	UF : 7, UT : 3,	CONFIG : 'F U T, 0, 0, 0',
	X =   -14.765  mm,	Y =   389.269  mm,	Z =     0.000  mm,
	W =  -167.358 deg,	P =     0.000 deg,	R =  -162.799 deg
};
P[92]{
   GP1:
	UF : 7, UT : 3,	CONFIG : 'F U T, 0, 0, 0',
	X =   -39.441  mm,	Y =   387.542  mm,	Z =     0.000  mm,
	W =  -167.357 deg,	P =     0.000 deg,	R =  -159.120 deg
};
P[93]{
   GP1:
	UF : 7, UT : 3,	CONFIG : 'F U T, 0, 0, 0',
	X =   -63.911  mm,	Y =   384.264  mm,	Z =     0.000  mm,
	W =  -167.357 deg,	P =     0.000 deg,	R =  -155.406 deg
};
P[94]{
   GP1:
	UF : 7, UT : 3,	CONFIG : 'F U T, 0, 0, 0',
	X =   -88.261  mm,	Y =   379.415  mm,	Z =     0.000  mm,
	W =  -167.357 deg,	P =    -0.001 deg,	R =  -151.728 deg
};
P[95]{
   GP1:
	UF : 7, UT : 3,	CONFIG : 'F U T, 0, 0, 0',
	X =  -112.432  mm,	Y =   372.971  mm,	Z =     0.000  mm,
	W =  -167.357 deg,	P =    -0.001 deg,	R =  -148.074 deg
};
P[96]{
   GP1:
	UF : 7, UT : 3,	CONFIG : 'F U T, 0, 0, 0',
	X =  -136.150  mm,	Y =   364.985  mm,	Z =     0.000  mm,
	W =  -167.357 deg,	P =    -0.002 deg,	R =  -144.425 deg
};
P[97]{
   GP1:
	UF : 7, UT : 3,	CONFIG : 'F U T, 0, 0, 0',
	X =  -159.308  mm,	Y =   355.490  mm,	Z =     0.000  mm,
	W =  -167.357 deg,	P =    -0.002 deg,	R =  -140.788 deg
};
P[98]{
   GP1:
	UF : 7, UT : 3,	CONFIG : 'F U T, 0, 0, 0',
	X =  -181.924  mm,	Y =   344.465  mm,	Z =     0.001  mm,
	W =  -167.357 deg,	P =    -0.003 deg,	R =  -137.121 deg
};
P[99]{
   GP1:
	UF : 7, UT : 3,	CONFIG : 'F U T, 0, 0, 0',
	X =  -201.161  mm,	Y =   333.583  mm,	Z =     0.001  mm,
	W =  -167.339 deg,	P =    -0.003 deg,	R =  -133.813 deg
};
P[100]{
   GP1:
	UF : 7, UT : 3,	CONFIG : 'F U T, 0, 0, 0',
	X =  -219.916  mm,	Y =   321.550  mm,	Z =     0.002  mm,
	W =  -167.321 deg,	P =    -0.006 deg,	R =  -130.535 deg
};
P[101]{
   GP1:
	UF : 7, UT : 3,	CONFIG : 'F U T, 0, 0, 0',
	X =  -238.197  mm,	Y =   308.239  mm,	Z =     0.003  mm,
	W =  -167.303 deg,	P =    -0.011 deg,	R =  -127.314 deg
};
P[102]{
   GP1:
	UF : 7, UT : 3,	CONFIG : 'F U T, 0, 0, 0',
	X =  -255.186  mm,	Y =   294.327  mm,	Z =     0.005  mm,
	W =  -167.286 deg,	P =    -0.018 deg,	R =  -123.984 deg
};
P[103]{
   GP1:
	UF : 7, UT : 3,	CONFIG : 'F U T, 0, 0, 0',
	X =  -271.779  mm,	Y =   279.082  mm,	Z =     0.007  mm,
	W =  -167.270 deg,	P =    -0.026 deg,	R =  -120.751 deg
};
P[104]{
   GP1:
	UF : 7, UT : 3,	CONFIG : 'F U T, 0, 0, 0',
	X =  -286.942  mm,	Y =   263.454  mm,	Z =     0.009  mm,
	W =  -167.255 deg,	P =    -0.037 deg,	R =  -117.421 deg
};
P[105]{
   GP1:
	UF : 7, UT : 3,	CONFIG : 'F U T, 0, 0, 0',
	X =  -298.890  mm,	Y =   249.815  mm,	Z =     0.013  mm,
	W =  -167.199 deg,	P =    -0.062 deg,	R =  -114.916 deg
};
P[106]{
   GP1:
	UF : 7, UT : 3,	CONFIG : 'F U T, 0, 0, 0',
	X =  -309.583  mm,	Y =   236.436  mm,	Z =     0.019  mm,
	W =  -167.149 deg,	P =    -0.092 deg,	R =  -112.269 deg
};
P[107]{
   GP1:
	UF : 7, UT : 3,	CONFIG : 'F U T, 0, 0, 0',
	X =  -320.386  mm,	Y =   221.580  mm,	Z =     0.036  mm,
	W =  -166.954 deg,	P =    -0.189 deg,	R =  -109.775 deg
};
P[108]{
   GP1:
	UF : 7, UT : 3,	CONFIG : 'F U T, 0, 0, 0',
	X =  -333.053  mm,	Y =   202.046  mm,	Z =     0.092  mm,
	W =  -166.266 deg,	P =    -0.517 deg,	R =  -106.161 deg
};
P[109]{
   GP1:
	UF : 7, UT : 3,	CONFIG : 'F U T, 0, 0, 0',
	X =  -342.020  mm,	Y =   186.464  mm,	Z =     0.185  mm,
	W =  -165.073 deg,	P =    -1.017 deg,	R =  -103.499 deg
};
P[110]{
   GP1:
	UF : 7, UT : 3,	CONFIG : 'F U T, 0, 0, 0',
	X =  -348.172  mm,	Y =   174.755  mm,	Z =     0.274  mm,
	W =  -163.892 deg,	P =    -1.242 deg,	R =  -101.659 deg
};
P[111]{
   GP1:
	UF : 7, UT : 3,	CONFIG : 'F U T, 0, 0, 0',
	X =  -352.609  mm,	Y =   165.627  mm,	Z =     0.302  mm,
	W =  -163.547 deg,	P =    -1.029 deg,	R =  -100.088 deg
};
P[112]{
   GP1:
	UF : 7, UT : 3,	CONFIG : 'F U T, 0, 0, 0',
	X =  -355.019  mm,	Y =   160.372  mm,	Z =     0.295  mm,
	W =  -163.656 deg,	P =    -0.836 deg,	R =   -99.364 deg
};
P[113]{
   GP1:
	UF : 7, UT : 3,	CONFIG : 'F U T, 0, 0, 0',
	X =  -362.143  mm,	Y =   143.583  mm,	Z =     0.211  mm,
	W =  -164.725 deg,	P =    -0.386 deg,	R =   -96.598 deg
};
P[114]{
   GP1:
	UF : 7, UT : 3,	CONFIG : 'F U T, 0, 0, 0',
	X =  -367.745  mm,	Y =   128.513  mm,	Z =     0.130  mm,
	W =  -165.767 deg,	P =    -0.146 deg,	R =   -94.271 deg
};
P[115]{
   GP1:
	UF : 7, UT : 3,	CONFIG : 'F U T, 0, 0, 0',
	X =  -371.689  mm,	Y =   116.596  mm,	Z =     0.074  mm,
	W =  -166.467 deg,	P =    -0.020 deg,	R =   -92.232 deg
};
P[116]{
   GP1:
	UF : 7, UT : 3,	CONFIG : 'F U T, 0, 0, 0',
	X =  -377.703  mm,	Y =    95.360  mm,	Z =     0.021  mm,
	W =  -167.125 deg,	P =     0.006 deg,	R =   -89.157 deg
};
P[117]{
   GP1:
	UF : 7, UT : 3,	CONFIG : 'F U T, 0, 0, 0',
	X =  -382.043  mm,	Y =    76.141  mm,	Z =     0.008  mm,
	W =  -167.278 deg,	P =    -0.003 deg,	R =   -86.170 deg
};
P[118]{
   GP1:
	UF : 7, UT : 3,	CONFIG : 'F U T, 0, 1, 0',
	X =  -385.149  mm,	Y =    58.405  mm,	Z =     0.004  mm,
	W =  -167.298 deg,	P =    -0.005 deg,	R =   -83.480 deg
};
P[119]{
   GP1:
	UF : 7, UT : 3,	CONFIG : 'F U T, 0, 1, 0',
	X =  -387.471  mm,	Y =    40.167  mm,	Z =     0.002  mm,
	W =  -167.319 deg,	P =    -0.005 deg,	R =   -80.834 deg
};
P[120]{
   GP1:
	UF : 7, UT : 3,	CONFIG : 'F U T, 0, 1, 0',
	X =  -388.901  mm,	Y =    22.351  mm,	Z =     0.001  mm,
	W =  -167.339 deg,	P =    -0.003 deg,	R =   -78.124 deg
};
P[121]{
   GP1:
	UF : 7, UT : 3,	CONFIG : 'F U T, 0, 1, 0',
	X =  -389.566  mm,	Y =     0.000  mm,	Z =     0.000  mm,
	W =  -167.363 deg,	P =     0.002 deg,	R =   -75.581 deg
};
P[122]{
   GP1:
	UF : 7, UT : 3,	CONFIG : 'F U T, 0, 1, 0',
	X =  -389.566  mm,	Y =     0.000  mm,	Z =     0.000  mm,
	W =  -167.363 deg,	P =     0.002 deg,	R =   -75.581 deg
};
P[123]{
   GP1:
	UF : 7, UT : 3,	CONFIG : 'F U T, 0, 1, 0',
	X =  -389.566  mm,	Y =     0.000  mm,	Z =     0.000  mm,
	W =  -167.363 deg,	P =     0.002 deg,	R =   -75.581 deg
};
P[124]{
   GP1:
	UF : 7, UT : 3,	CONFIG : 'F U T, 0, 1, 0',
	X =  -389.566  mm,	Y =     0.000  mm,	Z =     0.000  mm,
	W =  -167.363 deg,	P =     0.002 deg,	R =   -75.581 deg
};
P[125]{
   GP1:
	UF : 7, UT : 3,	CONFIG : 'F U T, 0, 1, 0',
	X =  -386.431  mm,	Y =     0.000  mm,	Z =     0.000  mm,
	W =  -167.363 deg,	P =     0.004 deg,	R =   -75.580 deg
};
P[126]{
   GP1:
	UF : 7, UT : 3,	CONFIG : 'F U T, 0, 1, 0',
	X =  -386.431  mm,	Y =     0.000  mm,	Z =     0.000  mm,
	W =  -167.363 deg,	P =     0.004 deg,	R =   -75.580 deg
};
P[127]{
   GP1:
	UF : 7, UT : 3,	CONFIG : 'F U T, 0, 1, 0',
	X =  -386.431  mm,	Y =     0.000  mm,	Z =     0.000  mm,
	W =  -167.363 deg,	P =     0.004 deg,	R =   -75.580 deg
};
P[128]{
   GP1:
	UF : 7, UT : 3,	CONFIG : 'F U T, 0, 1, 0',
	X =  -386.431  mm,	Y =     0.000  mm,	Z =     0.000  mm,
	W =  -167.363 deg,	P =     0.004 deg,	R =   -75.580 deg
};
P[129]{
   GP1:
	UF : 7, UT : 3,	CONFIG : 'F U T, 0, 1, 0',
	X =  -385.728  mm,	Y =    22.980  mm,	Z =     0.002  mm,
	W =  -167.343 deg,	P =     0.005 deg,	R =   -78.237 deg
};
P[130]{
   GP1:
	UF : 7, UT : 3,	CONFIG : 'F U T, 0, 1, 0',
	X =  -384.186  mm,	Y =    41.494  mm,	Z =     0.003  mm,
	W =  -167.327 deg,	P =     0.008 deg,	R =   -81.052 deg
};
P[131]{
   GP1:
	UF : 7, UT : 3,	CONFIG : 'F U T, 0, 1, 0',
	X =  -381.745  mm,	Y =    59.946  mm,	Z =     0.006  mm,
	W =  -167.311 deg,	P =     0.013 deg,	R =   -83.888 deg
};
P[132]{
   GP1:
	UF : 7, UT : 3,	CONFIG : 'F U T, 0, 0, 0',
	X =  -378.435  mm,	Y =    78.139  mm,	Z =     0.013  mm,
	W =  -167.296 deg,	P =     0.019 deg,	R =   -86.709 deg
};
P[133]{
   GP1:
	UF : 7, UT : 3,	CONFIG : 'F U T, 0, 0, 0',
	X =  -374.220  mm,	Y =    96.296  mm,	Z =     0.035  mm,
	W =  -167.174 deg,	P =     0.071 deg,	R =   -89.379 deg
};
P[134]{
   GP1:
	UF : 7, UT : 3,	CONFIG : 'F U T, 0, 0, 0',
	X =  -368.383  mm,	Y =   116.679  mm,	Z =     0.123  mm,
	W =  -166.585 deg,	P =     0.174 deg,	R =   -92.458 deg
};
P[135]{
   GP1:
	UF : 7, UT : 3,	CONFIG : 'F U T, 0, 0, 0',
	X =  -364.953  mm,	Y =   127.010  mm,	Z =     0.203  mm,
	W =  -166.017 deg,	P =     0.117 deg,	R =   -94.184 deg
};
P[136]{
   GP1:
	UF : 7, UT : 3,	CONFIG : 'F U T, 0, 0, 0',
	X =  -359.305  mm,	Y =   142.216  mm,	Z =     0.344  mm,
	W =  -165.061 deg,	P =    -0.074 deg,	R =   -96.543 deg
};
P[137]{
   GP1:
	UF : 7, UT : 3,	CONFIG : 'F U T, 0, 0, 0',
	X =  -352.423  mm,	Y =   158.543  mm,	Z =     0.487  mm,
	W =  -164.062 deg,	P =    -0.561 deg,	R =   -99.206 deg
};
P[138]{
   GP1:
	UF : 7, UT : 3,	CONFIG : 'F U T, 0, 0, 0',
	X =  -347.882  mm,	Y =   168.243  mm,	Z =     0.505  mm,
	W =  -163.926 deg,	P =    -1.110 deg,	R =  -100.804 deg
};
P[139]{
   GP1:
	UF : 7, UT : 3,	CONFIG : 'F U T, 0, 0, 0',
	X =  -343.610  mm,	Y =   176.790  mm,	Z =     0.432  mm,
	W =  -164.462 deg,	P =    -1.446 deg,	R =  -102.231 deg
};
P[140]{
   GP1:
	UF : 7, UT : 3,	CONFIG : 'F U T, 0, 0, 0',
	X =  -337.864  mm,	Y =   187.540  mm,	Z =     0.283  mm,
	W =  -165.514 deg,	P =    -1.149 deg,	R =  -103.973 deg
};
P[141]{
   GP1:
	UF : 7, UT : 3,	CONFIG : 'F U T, 0, 0, 0',
	X =  -329.121  mm,	Y =   202.489  mm,	Z =     0.139  mm,
	W =  -166.523 deg,	P =    -0.578 deg,	R =  -106.538 deg
};
P[142]{
   GP1:
	UF : 7, UT : 3,	CONFIG : 'F U T, 0, 0, 0',
	X =  -316.177  mm,	Y =   222.138  mm,	Z =     0.052  mm,
	W =  -167.084 deg,	P =    -0.195 deg,	R =  -109.921 deg
};
P[143]{
   GP1:
	UF : 7, UT : 3,	CONFIG : 'F U T, 0, 0, 0',
	X =  -304.752  mm,	Y =   237.588  mm,	Z =     0.027  mm,
	W =  -167.224 deg,	P =    -0.083 deg,	R =  -112.856 deg
};
P[144]{
   GP1:
	UF : 7, UT : 3,	CONFIG : 'F U T, 0, 0, 0',
	X =  -291.236  mm,	Y =   253.957  mm,	Z =     0.017  mm,
	W =  -167.254 deg,	P =    -0.055 deg,	R =  -116.039 deg
};
P[145]{
   GP1:
	UF : 7, UT : 3,	CONFIG : 'F U T, 0, 0, 0',
	X =  -276.686  mm,	Y =   269.748  mm,	Z =     0.013  mm,
	W =  -167.286 deg,	P =    -0.031 deg,	R =  -119.186 deg
};
P[146]{
   GP1:
	UF : 7, UT : 3,	CONFIG : 'F U T, 0, 0, 0',
	X =  -258.933  mm,	Y =   286.828  mm,	Z =     0.009  mm,
	W =  -167.297 deg,	P =    -0.022 deg,	R =  -122.790 deg
};
P[147]{
   GP1:
	UF : 7, UT : 3,	CONFIG : 'F U T, 0, 0, 0',
	X =  -240.334  mm,	Y =   302.578  mm,	Z =     0.006  mm,
	W =  -167.309 deg,	P =    -0.014 deg,	R =  -126.419 deg
};
P[148]{
   GP1:
	UF : 7, UT : 3,	CONFIG : 'F U T, 0, 0, 0',
	X =  -221.095  mm,	Y =   316.905  mm,	Z =     0.003  mm,
	W =  -167.321 deg,	P =    -0.009 deg,	R =  -130.112 deg
};
P[149]{
   GP1:
	UF : 7, UT : 3,	CONFIG : 'F U T, 0, 0, 0',
	X =  -200.765  mm,	Y =   330.162  mm,	Z =     0.002  mm,
	W =  -167.334 deg,	P =    -0.005 deg,	R =  -133.760 deg
};
P[150]{
   GP1:
	UF : 7, UT : 3,	CONFIG : 'F U T, 0, 0, 0',
	X =  -179.346  mm,	Y =   342.277  mm,	Z =     0.001  mm,
	W =  -167.347 deg,	P =    -0.002 deg,	R =  -137.374 deg
};
P[151]{
   GP1:
	UF : 7, UT : 3,	CONFIG : 'F U T, 0, 0, 0',
	X =  -157.102  mm,	Y =   353.047  mm,	Z =     0.001  mm,
	W =  -167.361 deg,	P =    -0.001 deg,	R =  -140.991 deg
};
P[152]{
   GP1:
	UF : 7, UT : 3,	CONFIG : 'F U T, 0, 0, 0',
	X =  -134.730  mm,	Y =   362.181  mm,	Z =     0.000  mm,
	W =  -167.361 deg,	P =    -0.001 deg,	R =  -144.507 deg
};
P[153]{
   GP1:
	UF : 7, UT : 3,	CONFIG : 'F U T, 0, 0, 0',
	X =  -111.889  mm,	Y =   369.863  mm,	Z =     0.000  mm,
	W =  -167.361 deg,	P =    -0.001 deg,	R =  -148.052 deg
};
P[154]{
   GP1:
	UF : 7, UT : 3,	CONFIG : 'F U T, 0, 0, 0',
	X =   -88.772  mm,	Y =   376.073  mm,	Z =     0.000  mm,
	W =  -167.361 deg,	P =    -0.001 deg,	R =  -151.635 deg
};
P[155]{
   GP1:
	UF : 7, UT : 3,	CONFIG : 'F U T, 0, 0, 0',
	X =   -65.616  mm,	Y =   380.803  mm,	Z =     0.000  mm,
	W =  -167.361 deg,	P =    -0.001 deg,	R =  -155.190 deg
};
P[156]{
   GP1:
	UF : 7, UT : 3,	CONFIG : 'F U T, 0, 0, 0',
	X =   -41.878  mm,	Y =   384.144  mm,	Z =     0.000  mm,
	W =  -167.361 deg,	P =     0.000 deg,	R =  -158.763 deg
};
P[157]{
   GP1:
	UF : 7, UT : 3,	CONFIG : 'F U T, 0, 0, 0',
	X =   -17.843  mm,	Y =   386.005  mm,	Z =     0.000  mm,
	W =  -167.361 deg,	P =     0.000 deg,	R =  -162.262 deg
};
P[158]{
   GP1:
	UF : 7, UT : 3,	CONFIG : 'F U T, 0, 0, 0',
	X =     6.524  mm,	Y =   386.359  mm,	Z =     0.000  mm,
	W =  -167.361 deg,	P =     0.000 deg,	R =  -165.807 deg
};
P[159]{
   GP1:
	UF : 7, UT : 3,	CONFIG : 'F U T, 0, 0, 0',
	X =    29.761  mm,	Y =   385.261  mm,	Z =     0.000  mm,
	W =  -167.361 deg,	P =     0.000 deg,	R =  -169.395 deg
};
P[160]{
   GP1:
	UF : 7, UT : 3,	CONFIG : 'F U T, 0, 0, 0',
	X =    53.260  mm,	Y =   382.727  mm,	Z =     0.000  mm,
	W =  -167.361 deg,	P =     0.000 deg,	R =  -172.963 deg
};
P[161]{
   GP1:
	UF : 7, UT : 3,	CONFIG : 'F U T, 0, 0, 0',
	X =    76.985  mm,	Y =   378.676  mm,	Z =     0.000  mm,
	W =  -167.361 deg,	P =     0.000 deg,	R =  -176.454 deg
};
P[162]{
   GP1:
	UF : 7, UT : 3,	CONFIG : 'F U T, 0, 0, 0',
	X =   100.333  mm,	Y =   373.172  mm,	Z =     0.000  mm,
	W =  -167.362 deg,	P =     0.000 deg,	R =  -179.957 deg
};
P[163]{
   GP1:
	UF : 7, UT : 3,	CONFIG : 'F U T, 0, 0, 0',
	X =   123.278  mm,	Y =   366.220  mm,	Z =     0.000  mm,
	W =  -167.362 deg,	P =     0.000 deg,	R =   176.516 deg
};
P[164]{
   GP1:
	UF : 7, UT : 3,	CONFIG : 'F U T, 0, 0, 0',
	X =   145.657  mm,	Y =   357.904  mm,	Z =     0.000  mm,
	W =  -167.362 deg,	P =     0.001 deg,	R =   172.960 deg
};
P[165]{
   GP1:
	UF : 7, UT : 3,	CONFIG : 'F U T, 0, 0, 0',
	X =   167.245  mm,	Y =   348.350  mm,	Z =     0.000  mm,
	W =  -167.362 deg,	P =     0.001 deg,	R =   169.347 deg
};
P[166]{
   GP1:
	UF : 7, UT : 3,	CONFIG : 'F U T, 0, 0, 0',
	X =   188.544  mm,	Y =   337.300  mm,	Z =     0.000  mm,
	W =  -167.362 deg,	P =     0.001 deg,	R =   165.827 deg
};
P[167]{
   GP1:
	UF : 7, UT : 3,	CONFIG : 'F U T, 0, 0, 0',
	X =   209.202  mm,	Y =   324.888  mm,	Z =     0.000  mm,
	W =  -167.362 deg,	P =     0.001 deg,	R =   162.330 deg
};
P[168]{
   GP1:
	UF : 7, UT : 3,	CONFIG : 'F U T, 0, 0, 0',
	X =   228.849  mm,	Y =   311.357  mm,	Z =     0.000  mm,
	W =  -167.362 deg,	P =     0.001 deg,	R =   158.779 deg
};
P[169]{
   GP1:
	UF : 7, UT : 3,	CONFIG : 'F U T, 0, 0, 0',
	X =   247.262  mm,	Y =   296.940  mm,	Z =     0.000  mm,
	W =  -167.362 deg,	P =     0.001 deg,	R =   155.200 deg
};
P[170]{
   GP1:
	UF : 7, UT : 3,	CONFIG : 'F U T, 0, 0, 0',
	X =   265.119  mm,	Y =   281.126  mm,	Z =     0.000  mm,
	W =  -167.363 deg,	P =     0.001 deg,	R =   151.683 deg
};
P[171]{
   GP1:
	UF : 7, UT : 3,	CONFIG : 'F U T, 0, 0, 0',
	X =   282.118  mm,	Y =   264.074  mm,	Z =     0.000  mm,
	W =  -167.363 deg,	P =     0.001 deg,	R =   148.165 deg
};
P[172]{
   GP1:
	UF : 7, UT : 3,	CONFIG : 'F U T, 0, 0, 0',
	X =   297.978  mm,	Y =   246.026  mm,	Z =     0.000  mm,
	W =  -167.363 deg,	P =     0.001 deg,	R =   144.655 deg
};
P[173]{
   GP1:
	UF : 7, UT : 3,	CONFIG : 'F U T, 0, 0, 0',
	X =   312.587  mm,	Y =   227.159  mm,	Z =     0.000  mm,
	W =  -167.363 deg,	P =     0.001 deg,	R =   141.125 deg
};
P[174]{
   GP1:
	UF : 7, UT : 3,	CONFIG : 'F U T, 0, 0, 0',
	X =   325.799  mm,	Y =   207.774  mm,	Z =     0.000  mm,
	W =  -167.363 deg,	P =     0.001 deg,	R =   137.537 deg
};
P[175]{
   GP1:
	UF : 7, UT : 3,	CONFIG : 'F U T, 0, 0, 0',
	X =   337.939  mm,	Y =   187.391  mm,	Z =     0.000  mm,
	W =  -167.363 deg,	P =     0.001 deg,	R =   134.013 deg
};
P[176]{
   GP1:
	UF : 7, UT : 3,	CONFIG : 'F U T, 0, 0, 0',
	X =   348.968  mm,	Y =   165.953  mm,	Z =     0.000  mm,
	W =  -167.363 deg,	P =     0.000 deg,	R =   130.515 deg
};
P[177]{
   GP1:
	UF : 7, UT : 3,	CONFIG : 'F U T, 0, 0, 0',
	X =   358.674  mm,	Y =   143.772  mm,	Z =     0.000  mm,
	W =  -167.363 deg,	P =     0.000 deg,	R =   126.963 deg
};
P[178]{
   GP1:
	UF : 7, UT : 3,	CONFIG : 'F U T, 0, 0, 0',
	X =   366.735  mm,	Y =   121.727  mm,	Z =     0.000  mm,
	W =  -167.363 deg,	P =     0.000 deg,	R =   123.366 deg
};
P[179]{
   GP1:
	UF : 7, UT : 3,	CONFIG : 'F U T, 0, 0, 0',
	X =   373.543  mm,	Y =    98.899  mm,	Z =     0.000  mm,
	W =  -167.363 deg,	P =     0.000 deg,	R =   119.795 deg
};
P[180]{
   GP1:
	UF : 7, UT : 3,	CONFIG : 'F U T, 0, 0, 0',
	X =   379.011  mm,	Y =    75.341  mm,	Z =     0.000  mm,
	W =  -167.363 deg,	P =     0.000 deg,	R =   116.250 deg
};
P[181]{
   GP1:
	UF : 7, UT : 3,	CONFIG : 'F U T, 0, 0, 0',
	X =   382.979  mm,	Y =    51.499  mm,	Z =     0.000  mm,
	W =  -167.363 deg,	P =     0.000 deg,	R =   112.726 deg
};
P[182]{
   GP1:
	UF : 7, UT : 3,	CONFIG : 'F U T, 0, 0, 0',
	X =   385.447  mm,	Y =    27.385  mm,	Z =     0.000  mm,
	W =  -167.364 deg,	P =     0.000 deg,	R =   109.204 deg
};
P[183]{
   GP1:
	UF : 7, UT : 3,	CONFIG : 'F U T, 0, 0, 0',
	X =   386.431  mm,	Y =     0.000  mm,	Z =     0.000  mm,
	W =  -167.364 deg,	P =     0.000 deg,	R =   105.687 deg
};
P[184]{
   GP1:
	UF : 7, UT : 3,	CONFIG : 'F U T, 0, 0, 0',
	X =   386.431  mm,	Y =     0.000  mm,	Z =     0.000  mm,
	W =  -167.364 deg,	P =     0.000 deg,	R =   105.687 deg
};
P[185]{
   GP1:
	UF : 7, UT : 3,	CONFIG : 'F U T, 0, 0, 0',
	X =   386.431  mm,	Y =     0.000  mm,	Z =     0.000  mm,
	W =  -167.364 deg,	P =     0.000 deg,	R =   105.687 deg
};
P[186]{
   GP1:
	UF : 7, UT : 3,	CONFIG : 'F U T, 0, 0, 0',
	X =   386.431  mm,	Y =     0.000  mm,	Z =     0.000  mm,
	W =  -167.364 deg,	P =     0.000 deg,	R =   105.687 deg
};
P[187]{
   GP1:
	UF : 7, UT : 3,	CONFIG : 'F U T, 0, 0, 0',
	X =   383.297  mm,	Y =     0.000  mm,	Z =     0.000  mm,
	W =  -167.364 deg,	P =     0.000 deg,	R =   105.687 deg
};
P[188]{
   GP1:
	UF : 7, UT : 3,	CONFIG : 'F U T, 0, 0, 0',
	X =   383.297  mm,	Y =     0.000  mm,	Z =     0.000  mm,
	W =  -167.364 deg,	P =     0.000 deg,	R =   105.687 deg
};
P[189]{
   GP1:
	UF : 7, UT : 3,	CONFIG : 'F U T, 0, 0, 0',
	X =   383.297  mm,	Y =     0.000  mm,	Z =     0.000  mm,
	W =  -167.364 deg,	P =     0.000 deg,	R =   105.687 deg
};
P[190]{
   GP1:
	UF : 7, UT : 3,	CONFIG : 'F U T, 0, 0, 0',
	X =   383.297  mm,	Y =     0.000  mm,	Z =     0.000  mm,
	W =  -167.364 deg,	P =     0.000 deg,	R =   105.687 deg
};
P[191]{
   GP1:
	UF : 7, UT : 3,	CONFIG : 'F U T, 0, 0, 0',
	X =   382.233  mm,	Y =    28.263  mm,	Z =     0.000  mm,
	W =  -167.364 deg,	P =     0.000 deg,	R =   109.413 deg
};
P[192]{
   GP1:
	UF : 7, UT : 3,	CONFIG : 'F U T, 0, 0, 0',
	X =   379.557  mm,	Y =    53.272  mm,	Z =     0.000  mm,
	W =  -167.364 deg,	P =     0.000 deg,	R =   113.113 deg
};
P[193]{
   GP1:
	UF : 7, UT : 3,	CONFIG : 'F U T, 0, 0, 0',
	X =   375.303  mm,	Y =    77.800  mm,	Z =     0.000  mm,
	W =  -167.364 deg,	P =    -0.001 deg,	R =   116.833 deg
};
P[194]{
   GP1:
	UF : 7, UT : 3,	CONFIG : 'F U T, 0, 0, 0',
	X =   369.435  mm,	Y =   102.116  mm,	Z =     0.000  mm,
	W =  -167.364 deg,	P =    -0.001 deg,	R =   120.571 deg
};
P[195]{
   GP1:
	UF : 7, UT : 3,	CONFIG : 'F U T, 0, 0, 0',
	X =   361.971  mm,	Y =   126.046  mm,	Z =     0.000  mm,
	W =  -167.364 deg,	P =    -0.001 deg,	R =   124.293 deg
};
P[196]{
   GP1:
	UF : 7, UT : 3,	CONFIG : 'F U T, 0, 0, 0',
	X =   352.945  mm,	Y =   149.476  mm,	Z =     0.000  mm,
	W =  -167.364 deg,	P =    -0.001 deg,	R =   128.040 deg
};
P[197]{
   GP1:
	UF : 7, UT : 3,	CONFIG : 'F U T, 0, 0, 0',
	X =   342.445  mm,	Y =   172.178  mm,	Z =     0.000  mm,
	W =  -167.364 deg,	P =    -0.001 deg,	R =   131.767 deg
};
P[198]{
   GP1:
	UF : 7, UT : 3,	CONFIG : 'F U T, 0, 0, 0',
	X =   330.428  mm,	Y =   194.250  mm,	Z =     0.000  mm,
	W =  -167.364 deg,	P =    -0.001 deg,	R =   135.511 deg
};
P[199]{
   GP1:
	UF : 7, UT : 3,	CONFIG : 'F U T, 0, 0, 0',
	X =   317.027  mm,	Y =   215.424  mm,	Z =     0.000  mm,
	W =  -167.364 deg,	P =    -0.001 deg,	R =   139.239 deg
};
P[200]{
   GP1:
	UF : 7, UT : 3,	CONFIG : 'F U T, 0, 0, 0',
	X =   302.327  mm,	Y =   235.598  mm,	Z =     0.000  mm,
	W =  -167.365 deg,	P =    -0.001 deg,	R =   142.962 deg
};
P[201]{
   GP1:
	UF : 7, UT : 3,	CONFIG : 'F U T, 0, 0, 0',
	X =   286.286  mm,	Y =   254.853  mm,	Z =     0.000  mm,
	W =  -167.365 deg,	P =    -0.001 deg,	R =   146.664 deg
};
P[202]{
   GP1:
	UF : 7, UT : 3,	CONFIG : 'F U T, 0, 0, 0',
	X =   269.131  mm,	Y =   272.899  mm,	Z =     0.000  mm,
	W =  -167.365 deg,	P =    -0.001 deg,	R =   150.376 deg
};
P[203]{
   GP1:
	UF : 7, UT : 3,	CONFIG : 'F U T, 0, 0, 0',
	X =   250.694  mm,	Y =   289.925  mm,	Z =     0.000  mm,
	W =  -167.365 deg,	P =    -0.001 deg,	R =   154.094 deg
};
P[204]{
   GP1:
	UF : 7, UT : 3,	CONFIG : 'F U T, 0, 0, 0',
	X =   231.382  mm,	Y =   305.556  mm,	Z =     0.000  mm,
	W =  -167.365 deg,	P =    -0.001 deg,	R =   157.816 deg
};
P[205]{
   GP1:
	UF : 7, UT : 3,	CONFIG : 'F U T, 0, 0, 0',
	X =   211.214  mm,	Y =   319.828  mm,	Z =     0.000  mm,
	W =  -167.365 deg,	P =    -0.001 deg,	R =   161.551 deg
};
P[206]{
   GP1:
	UF : 7, UT : 3,	CONFIG : 'F U T, 0, 0, 0',
	X =   190.290  mm,	Y =   332.701  mm,	Z =     0.000  mm,
	W =  -167.365 deg,	P =     0.000 deg,	R =   165.307 deg
};
P[207]{
   GP1:
	UF : 7, UT : 3,	CONFIG : 'F U T, 0, 0, 0',
	X =   168.391  mm,	Y =   344.303  mm,	Z =     0.000  mm,
	W =  -167.365 deg,	P =     0.000 deg,	R =   169.046 deg
};
P[208]{
   GP1:
	UF : 7, UT : 3,	CONFIG : 'F U T, 0, 0, 0',
	X =   145.892  mm,	Y =   354.424  mm,	Z =     0.000  mm,
	W =  -167.366 deg,	P =     0.000 deg,	R =   172.806 deg
};
P[209]{
   GP1:
	UF : 7, UT : 3,	CONFIG : 'F U T, 0, 0, 0',
	X =   122.424  mm,	Y =   363.199  mm,	Z =     0.000  mm,
	W =  -167.366 deg,	P =     0.000 deg,	R =   176.501 deg
};
P[210]{
   GP1:
	UF : 7, UT : 3,	CONFIG : 'F U T, 0, 0, 0',
	X =    98.612  mm,	Y =   370.378  mm,	Z =     0.000  mm,
	W =  -167.366 deg,	P =     0.000 deg,	R =  -179.791 deg
};
P[211]{
   GP1:
	UF : 7, UT : 3,	CONFIG : 'F U T, 0, 0, 0',
	X =    74.337  mm,	Y =   376.007  mm,	Z =     0.000  mm,
	W =  -167.366 deg,	P =     0.000 deg,	R =  -176.079 deg
};
P[212]{
   GP1:
	UF : 7, UT : 3,	CONFIG : 'F U T, 0, 0, 0',
	X =    49.660  mm,	Y =   380.060  mm,	Z =     0.000  mm,
	W =  -167.366 deg,	P =     0.000 deg,	R =  -172.343 deg
};
P[213]{
   GP1:
	UF : 7, UT : 3,	CONFIG : 'F U T, 0, 0, 0',
	X =    24.688  mm,	Y =   382.498  mm,	Z =     0.000  mm,
	W =  -167.366 deg,	P =     0.001 deg,	R =  -168.608 deg
};
P[214]{
   GP1:
	UF : 7, UT : 3,	CONFIG : 'F U T, 0, 0, 0',
	X =    -0.526  mm,	Y =   383.297  mm,	Z =     0.000  mm,
	W =  -167.366 deg,	P =     0.001 deg,	R =  -164.843 deg
};
P[215]{
   GP1:
	UF : 7, UT : 3,	CONFIG : 'F U T, 0, 0, 0',
	X =   -25.627  mm,	Y =   382.438  mm,	Z =     0.000  mm,
	W =  -167.366 deg,	P =     0.001 deg,	R =  -161.103 deg
};
P[216]{
   GP1:
	UF : 7, UT : 3,	CONFIG : 'F U T, 0, 0, 0',
	X =   -50.599  mm,	Y =   379.941  mm,	Z =     0.000  mm,
	W =  -167.366 deg,	P =     0.001 deg,	R =  -157.368 deg
};
P[217]{
   GP1:
	UF : 7, UT : 3,	CONFIG : 'F U T, 0, 0, 0',
	X =   -75.258  mm,	Y =   375.827  mm,	Z =     0.000  mm,
	W =  -167.366 deg,	P =     0.001 deg,	R =  -153.642 deg
};
P[218]{
   GP1:
	UF : 7, UT : 3,	CONFIG : 'F U T, 0, 0, 0',
	X =   -99.688  mm,	Y =   370.099  mm,	Z =     0.000  mm,
	W =  -167.366 deg,	P =     0.002 deg,	R =  -149.920 deg
};
P[219]{
   GP1:
	UF : 7, UT : 3,	CONFIG : 'F U T, 0, 0, 0',
	X =  -123.640  mm,	Y =   362.796  mm,	Z =     0.000  mm,
	W =  -167.366 deg,	P =     0.002 deg,	R =  -146.192 deg
};
P[220]{
   GP1:
	UF : 7, UT : 3,	CONFIG : 'F U T, 0, 0, 0',
	X =  -147.118  mm,	Y =   353.923  mm,	Z =     0.001  mm,
	W =  -167.366 deg,	P =     0.002 deg,	R =  -142.459 deg
};
P[221]{
   GP1:
	UF : 7, UT : 3,	CONFIG : 'F U T, 0, 0, 0',
	X =  -169.859  mm,	Y =   343.585  mm,	Z =     0.001  mm,
	W =  -167.366 deg,	P =     0.002 deg,	R =  -138.737 deg
};
P[222]{
   GP1:
	UF : 7, UT : 3,	CONFIG : 'F U T, 0, 0, 0',
	X =  -191.914  mm,	Y =   331.769  mm,	Z =     0.002  mm,
	W =  -167.366 deg,	P =     0.003 deg,	R =  -135.016 deg
};
P[223]{
   GP1:
	UF : 7, UT : 3,	CONFIG : 'F U T, 0, 0, 0',
	X =  -212.973  mm,	Y =   318.658  mm,	Z =     0.004  mm,
	W =  -167.366 deg,	P =     0.003 deg,	R =  -131.274 deg
};
P[224]{
   GP1:
	UF : 7, UT : 3,	CONFIG : 'F U T, 0, 0, 0',
	X =  -233.097  mm,	Y =   304.246  mm,	Z =     0.007  mm,
	W =  -167.366 deg,	P =     0.003 deg,	R =  -127.533 deg
};
P[225]{
   GP1:
	UF : 7, UT : 3,	CONFIG : 'F U T, 0, 0, 0',
	X =  -252.177  mm,	Y =   288.629  mm,	Z =     0.011  mm,
	W =  -167.366 deg,	P =     0.003 deg,	R =  -123.759 deg
};
P[226]{
   GP1:
	UF : 7, UT : 3,	CONFIG : 'F U T, 0, 0, 0',
	X =  -270.274  mm,	Y =   271.758  mm,	Z =     0.016  mm,
	W =  -167.365 deg,	P =     0.003 deg,	R =  -120.000 deg
};
P[227]{
   GP1:
	UF : 7, UT : 3,	CONFIG : 'F U T, 0, 0, 0',
	X =  -287.342  mm,	Y =   253.645  mm,	Z =     0.021  mm,
	W =  -167.365 deg,	P =     0.004 deg,	R =  -116.239 deg
};
P[228]{
   GP1:
	UF : 7, UT : 3,	CONFIG : 'F U T, 0, 0, 0',
	X =  -303.326  mm,	Y =   234.299  mm,	Z =     0.036  mm,
	W =  -167.365 deg,	P =     0.004 deg,	R =  -112.515 deg
};
P[229]{
   GP1:
	UF : 7, UT : 3,	CONFIG : 'F U T, 0, 0, 0',
	X =  -317.986  mm,	Y =   213.987  mm,	Z =     0.093  mm,
	W =  -167.365 deg,	P =     0.004 deg,	R =  -108.787 deg
};
P[230]{
   GP1:
	UF : 7, UT : 3,	CONFIG : 'F U T, 0, 0, 0',
	X =  -331.281  mm,	Y =   192.780  mm,	Z =     0.285  mm,
	W =  -167.365 deg,	P =     0.004 deg,	R =  -105.083 deg
};
P[231]{
   GP1:
	UF : 7, UT : 3,	CONFIG : 'F U T, 0, 0, 0',
	X =  -343.068  mm,	Y =   170.974  mm,	Z =     0.661  mm,
	W =  -167.364 deg,	P =     0.004 deg,	R =  -101.432 deg
};
P[232]{
   GP1:
	UF : 7, UT : 3,	CONFIG : 'F U T, 0, 0, 0',
	X =  -353.037  mm,	Y =   149.295  mm,	Z =     0.567  mm,
	W =  -167.364 deg,	P =     0.005 deg,	R =   -97.857 deg
};
P[233]{
   GP1:
	UF : 7, UT : 3,	CONFIG : 'F U T, 0, 0, 0',
	X =  -362.015  mm,	Y =   125.930  mm,	Z =     0.265  mm,
	W =  -167.364 deg,	P =     0.005 deg,	R =   -94.148 deg
};
P[234]{
   GP1:
	UF : 7, UT : 3,	CONFIG : 'F U T, 0, 0, 0',
	X =  -369.456  mm,	Y =   102.041  mm,	Z =     0.064  mm,
	W =  -167.364 deg,	P =     0.005 deg,	R =   -90.448 deg
};
P[235]{
   GP1:
	UF : 7, UT : 3,	CONFIG : 'F U T, 0, 0, 0',
	X =  -375.311  mm,	Y =    77.762  mm,	Z =     0.015  mm,
	W =  -167.363 deg,	P =     0.005 deg,	R =   -86.714 deg
};
P[236]{
   GP1:
	UF : 7, UT : 3,	CONFIG : 'F U T, 0, 1, 0',
	X =  -379.567  mm,	Y =    53.206  mm,	Z =     0.006  mm,
	W =  -167.363 deg,	P =     0.005 deg,	R =   -82.995 deg
};
P[237]{
   GP1:
	UF : 7, UT : 3,	CONFIG : 'F U T, 0, 1, 0',
	X =  -382.236  mm,	Y =    28.229  mm,	Z =     0.003  mm,
	W =  -167.363 deg,	P =     0.005 deg,	R =   -79.296 deg
};
P[238]{
   GP1:
	UF : 7, UT : 3,	CONFIG : 'F U T, 0, 1, 0',
	X =  -383.297  mm,	Y =     0.000  mm,	Z =     0.000  mm,
	W =  -167.362 deg,	P =     0.005 deg,	R =   -75.580 deg
};
P[239]{
   GP1:
	UF : 7, UT : 3,	CONFIG : 'F U T, 0, 1, 0',
	X =  -383.297  mm,	Y =     0.000  mm,	Z =     0.000  mm,
	W =  -167.362 deg,	P =     0.005 deg,	R =   -75.580 deg
};
P[240]{
   GP1:
	UF : 7, UT : 3,	CONFIG : 'F U T, 0, 1, 0',
	X =  -383.297  mm,	Y =     0.000  mm,	Z =     0.000  mm,
	W =  -167.362 deg,	P =     0.005 deg,	R =   -75.580 deg
};
P[241]{
   GP1:
	UF : 7, UT : 3,	CONFIG : 'F U T, 0, 1, 0',
	X =  -383.297  mm,	Y =     0.000  mm,	Z =     0.000  mm,
	W =  -167.362 deg,	P =     0.005 deg,	R =   -75.580 deg
};
P[242]{
   GP1:
	UF : 7, UT : 3,	CONFIG : 'F U T, 0, 1, 0',
	X =  -380.163  mm,	Y =     0.000  mm,	Z =     0.000  mm,
	W =  -167.362 deg,	P =     0.006 deg,	R =   -75.580 deg
};
P[243]{
   GP1:
	UF : 7, UT : 3,	CONFIG : 'F U T, 0, 1, 0',
	X =  -380.163  mm,	Y =     0.000  mm,	Z =     0.000  mm,
	W =  -167.362 deg,	P =     0.006 deg,	R =   -75.580 deg
};
P[244]{
   GP1:
	UF : 7, UT : 3,	CONFIG : 'F U T, 0, 1, 0',
	X =  -380.163  mm,	Y =     0.000  mm,	Z =     0.000  mm,
	W =  -167.362 deg,	P =     0.006 deg,	R =   -75.580 deg
};
P[245]{
   GP1:
	UF : 7, UT : 3,	CONFIG : 'F U T, 0, 1, 0',
	X =  -380.163  mm,	Y =     0.000  mm,	Z =     0.000  mm,
	W =  -167.362 deg,	P =     0.006 deg,	R =   -75.580 deg
};
P[246]{
   GP1:
	UF : 7, UT : 3,	CONFIG : 'F U T, 0, 1, 0',
	X =  -379.097  mm,	Y =    28.176  mm,	Z =     0.003  mm,
	W =  -167.362 deg,	P =     0.006 deg,	R =   -79.288 deg
};
P[247]{
   GP1:
	UF : 7, UT : 3,	CONFIG : 'F U T, 0, 1, 0',
	X =  -376.436  mm,	Y =    52.973  mm,	Z =     0.007  mm,
	W =  -167.363 deg,	P =     0.006 deg,	R =   -82.994 deg
};
P[248]{
   GP1:
	UF : 7, UT : 3,	CONFIG : 'F U T, 0, 0, 0',
	X =  -372.196  mm,	Y =    77.348  mm,	Z =     0.016  mm,
	W =  -167.363 deg,	P =     0.006 deg,	R =   -86.711 deg
};
P[249]{
   GP1:
	UF : 7, UT : 3,	CONFIG : 'F U T, 0, 0, 0',
	X =  -366.389  mm,	Y =   101.359  mm,	Z =     0.070  mm,
	W =  -167.364 deg,	P =     0.006 deg,	R =   -90.458 deg
};
P[250]{
   GP1:
	UF : 7, UT : 3,	CONFIG : 'F U T, 0, 0, 0',
	X =  -359.057  mm,	Y =   124.878  mm,	Z =     0.312  mm,
	W =  -167.364 deg,	P =     0.006 deg,	R =   -94.157 deg
};
P[251]{
   GP1:
	UF : 7, UT : 3,	CONFIG : 'F U T, 0, 0, 0',
	X =  -350.130  mm,	Y =   148.106  mm,	Z =     0.686  mm,
	W =  -167.364 deg,	P =     0.005 deg,	R =   -97.867 deg
};
P[252]{
   GP1:
	UF : 7, UT : 3,	CONFIG : 'F U T, 0, 0, 0',
	X =  -340.338  mm,	Y =   169.426  mm,	Z =     0.827  mm,
	W =  -167.365 deg,	P =     0.005 deg,	R =  -101.400 deg
};
P[253]{
   GP1:
	UF : 7, UT : 3,	CONFIG : 'F U T, 0, 0, 0',
	X =  -328.877  mm,	Y =   190.676  mm,	Z =     0.365  mm,
	W =  -167.365 deg,	P =     0.005 deg,	R =  -105.036 deg
};
P[254]{
   GP1:
	UF : 7, UT : 3,	CONFIG : 'F U T, 0, 0, 0',
	X =  -315.774  mm,	Y =   211.655  mm,	Z =     0.115  mm,
	W =  -167.365 deg,	P =     0.005 deg,	R =  -108.714 deg
};
P[255]{
   GP1:
	UF : 7, UT : 3,	CONFIG : 'F U T, 0, 0, 0',
	X =  -301.199  mm,	Y =   231.921  mm,	Z =     0.042  mm,
	W =  -167.365 deg,	P =     0.005 deg,	R =  -112.426 deg
};
P[256]{
   GP1:
	UF : 7, UT : 3,	CONFIG : 'F U T, 0, 0, 0',
	X =  -285.524  mm,	Y =   250.965  mm,	Z =     0.025  mm,
	W =  -167.366 deg,	P =     0.004 deg,	R =  -116.182 deg
};
P[257]{
   GP1:
	UF : 7, UT : 3,	CONFIG : 'F U T, 0, 0, 0',
	X =  -268.792  mm,	Y =   268.809  mm,	Z =     0.019  mm,
	W =  -167.366 deg,	P =     0.004 deg,	R =  -119.948 deg
};
P[258]{
   GP1:
	UF : 7, UT : 3,	CONFIG : 'F U T, 0, 0, 0',
	X =  -250.935  mm,	Y =   285.550  mm,	Z =     0.014  mm,
	W =  -167.366 deg,	P =     0.004 deg,	R =  -123.705 deg
};
P[259]{
   GP1:
	UF : 7, UT : 3,	CONFIG : 'F U T, 0, 0, 0',
	X =  -231.937  mm,	Y =   301.187  mm,	Z =     0.008  mm,
	W =  -167.366 deg,	P =     0.004 deg,	R =  -127.456 deg
};
P[260]{
   GP1:
	UF : 7, UT : 3,	CONFIG : 'F U T, 0, 0, 0',
	X =  -211.688  mm,	Y =   315.751  mm,	Z =     0.004  mm,
	W =  -167.366 deg,	P =     0.003 deg,	R =  -131.184 deg
};
P[261]{
   GP1:
	UF : 7, UT : 3,	CONFIG : 'F U T, 0, 0, 0',
	X =  -190.558  mm,	Y =   328.938  mm,	Z =     0.002  mm,
	W =  -167.367 deg,	P =     0.003 deg,	R =  -134.906 deg
};
P[262]{
   GP1:
	UF : 7, UT : 3,	CONFIG : 'F U T, 0, 0, 0',
	X =  -168.649  mm,	Y =   340.695  mm,	Z =     0.001  mm,
	W =  -167.367 deg,	P =     0.003 deg,	R =  -138.652 deg
};
P[263]{
   GP1:
	UF : 7, UT : 3,	CONFIG : 'F U T, 0, 0, 0',
	X =  -146.049  mm,	Y =   350.978  mm,	Z =     0.001  mm,
	W =  -167.367 deg,	P =     0.002 deg,	R =  -142.400 deg
};
P[264]{
   GP1:
	UF : 7, UT : 3,	CONFIG : 'F U T, 0, 0, 0',
	X =  -122.942  mm,	Y =   359.721  mm,	Z =     0.000  mm,
	W =  -167.367 deg,	P =     0.002 deg,	R =  -146.126 deg
};
P[265]{
   GP1:
	UF : 7, UT : 3,	CONFIG : 'F U T, 0, 0, 0',
	X =   -99.282  mm,	Y =   366.956  mm,	Z =     0.000  mm,
	W =  -167.367 deg,	P =     0.002 deg,	R =  -149.836 deg
};
P[266]{
   GP1:
	UF : 7, UT : 3,	CONFIG : 'F U T, 0, 0, 0',
	X =   -75.057  mm,	Y =   372.668  mm,	Z =     0.000  mm,
	W =  -167.367 deg,	P =     0.002 deg,	R =  -153.566 deg
};
P[267]{
   GP1:
	UF : 7, UT : 3,	CONFIG : 'F U T, 0, 0, 0',
	X =   -50.438  mm,	Y =   376.794  mm,	Z =     0.000  mm,
	W =  -167.367 deg,	P =     0.001 deg,	R =  -157.317 deg
};
P[268]{
   GP1:
	UF : 7, UT : 3,	CONFIG : 'F U T, 0, 0, 0',
	X =   -25.660  mm,	Y =   379.292  mm,	Z =     0.000  mm,
	W =  -167.367 deg,	P =     0.001 deg,	R =  -161.055 deg
};
P[269]{
   GP1:
	UF : 7, UT : 3,	CONFIG : 'F U T, 0, 0, 0',
	X =    -0.782  mm,	Y =   380.160  mm,	Z =     0.000  mm,
	W =  -167.367 deg,	P =     0.001 deg,	R =  -164.794 deg
};
P[270]{
   GP1:
	UF : 7, UT : 3,	CONFIG : 'F U T, 0, 0, 0',
	X =    24.076  mm,	Y =   379.389  mm,	Z =     0.000  mm,
	W =  -167.367 deg,	P =     0.001 deg,	R =  -168.539 deg
};
P[271]{
   GP1:
	UF : 7, UT : 3,	CONFIG : 'F U T, 0, 0, 0',
	X =    48.777  mm,	Y =   377.006  mm,	Z =     0.000  mm,
	W =  -167.367 deg,	P =     0.000 deg,	R =  -172.247 deg
};
P[272]{
   GP1:
	UF : 7, UT : 3,	CONFIG : 'F U T, 0, 0, 0',
	X =    73.339  mm,	Y =   373.005  mm,	Z =     0.000  mm,
	W =  -167.366 deg,	P =     0.000 deg,	R =  -175.979 deg
};
P[273]{
   GP1:
	UF : 7, UT : 3,	CONFIG : 'F U T, 0, 0, 0',
	X =    97.338  mm,	Y =   367.473  mm,	Z =     0.000  mm,
	W =  -167.366 deg,	P =     0.000 deg,	R =  -179.706 deg
};
P[274]{
   GP1:
	UF : 7, UT : 3,	CONFIG : 'F U T, 0, 0, 0',
	X =   120.910  mm,	Y =   360.402  mm,	Z =     0.000  mm,
	W =  -167.366 deg,	P =     0.000 deg,	R =   176.507 deg
};
P[275]{
   GP1:
	UF : 7, UT : 3,	CONFIG : 'F U T, 0, 0, 0',
	X =   144.079  mm,	Y =   351.780  mm,	Z =     0.000  mm,
	W =  -167.366 deg,	P =     0.000 deg,	R =   172.783 deg
};
P[276]{
   GP1:
	UF : 7, UT : 3,	CONFIG : 'F U T, 0, 0, 0',
	X =   166.693  mm,	Y =   341.643  mm,	Z =     0.000  mm,
	W =  -167.366 deg,	P =     0.000 deg,	R =   169.038 deg
};
P[277]{
   GP1:
	UF : 7, UT : 3,	CONFIG : 'F U T, 0, 0, 0',
	X =   188.803  mm,	Y =   329.939  mm,	Z =     0.000  mm,
	W =  -167.366 deg,	P =    -0.001 deg,	R =   165.315 deg
};
P[278]{
   GP1:
	UF : 7, UT : 3,	CONFIG : 'F U T, 0, 0, 0',
	X =   209.781  mm,	Y =   317.017  mm,	Z =     0.000  mm,
	W =  -167.366 deg,	P =    -0.001 deg,	R =   161.576 deg
};
P[279]{
   GP1:
	UF : 7, UT : 3,	CONFIG : 'F U T, 0, 0, 0',
	X =   229.691  mm,	Y =   302.906  mm,	Z =     0.000  mm,
	W =  -167.365 deg,	P =    -0.001 deg,	R =   157.796 deg
};
P[280]{
   GP1:
	UF : 7, UT : 3,	CONFIG : 'F U T, 0, 0, 0',
	X =   248.802  mm,	Y =   287.416  mm,	Z =     0.000  mm,
	W =  -167.365 deg,	P =    -0.001 deg,	R =   154.081 deg
};
P[281]{
   GP1:
	UF : 7, UT : 3,	CONFIG : 'F U T, 0, 0, 0',
	X =   266.984  mm,	Y =   270.613  mm,	Z =     0.000  mm,
	W =  -167.365 deg,	P =    -0.001 deg,	R =   150.358 deg
};
P[282]{
   GP1:
	UF : 7, UT : 3,	CONFIG : 'F U T, 0, 0, 0',
	X =   284.072  mm,	Y =   252.621  mm,	Z =     0.000  mm,
	W =  -167.365 deg,	P =    -0.001 deg,	R =   146.661 deg
};
P[283]{
   GP1:
	UF : 7, UT : 3,	CONFIG : 'F U T, 0, 0, 0',
	X =   299.952  mm,	Y =   233.557  mm,	Z =     0.000  mm,
	W =  -167.365 deg,	P =    -0.001 deg,	R =   142.927 deg
};
P[284]{
   GP1:
	UF : 7, UT : 3,	CONFIG : 'F U T, 0, 0, 0',
	X =   314.565  mm,	Y =   213.461  mm,	Z =     0.000  mm,
	W =  -167.365 deg,	P =    -0.001 deg,	R =   139.198 deg
};
P[285]{
   GP1:
	UF : 7, UT : 3,	CONFIG : 'F U T, 0, 0, 0',
	X =   327.812  mm,	Y =   192.504  mm,	Z =     0.000  mm,
	W =  -167.364 deg,	P =    -0.001 deg,	R =   135.478 deg
};
P[286]{
   GP1:
	UF : 7, UT : 3,	CONFIG : 'F U T, 0, 0, 0',
	X =   339.719  mm,	Y =   170.609  mm,	Z =     0.000  mm,
	W =  -167.364 deg,	P =    -0.001 deg,	R =   131.742 deg
};
P[287]{
   GP1:
	UF : 7, UT : 3,	CONFIG : 'F U T, 0, 0, 0',
	X =   350.124  mm,	Y =   148.078  mm,	Z =     0.000  mm,
	W =  -167.364 deg,	P =    -0.001 deg,	R =   128.016 deg
};
P[288]{
   GP1:
	UF : 7, UT : 3,	CONFIG : 'F U T, 0, 0, 0',
	X =   359.021  mm,	Y =   124.970  mm,	Z =     0.000  mm,
	W =  -167.364 deg,	P =    -0.001 deg,	R =   124.302 deg
};
P[289]{
   GP1:
	UF : 7, UT : 3,	CONFIG : 'F U T, 0, 0, 0',
	X =   366.382  mm,	Y =   101.383  mm,	Z =     0.000  mm,
	W =  -167.364 deg,	P =    -0.001 deg,	R =   120.570 deg
};
P[290]{
   GP1:
	UF : 7, UT : 3,	CONFIG : 'F U T, 0, 0, 0',
	X =   372.168  mm,	Y =    77.482  mm,	Z =     0.000  mm,
	W =  -167.364 deg,	P =    -0.001 deg,	R =   116.839 deg
};
P[291]{
   GP1:
	UF : 7, UT : 3,	CONFIG : 'F U T, 0, 0, 0',
	X =   376.438  mm,	Y =    52.971  mm,	Z =     0.000  mm,
	W =  -167.364 deg,	P =    -0.001 deg,	R =   113.130 deg
};
P[292]{
   GP1:
	UF : 7, UT : 3,	CONFIG : 'F U T, 0, 0, 0',
	X =   379.098  mm,	Y =    28.167  mm,	Z =     0.000  mm,
	W =  -167.364 deg,	P =     0.000 deg,	R =   109.392 deg
};
P[293]{
   GP1:
	UF : 7, UT : 3,	CONFIG : 'F U T, 0, 0, 0',
	X =   380.163  mm,	Y =     0.000  mm,	Z =     0.000  mm,
	W =  -167.364 deg,	P =     0.000 deg,	R =   105.687 deg
};
P[294]{
   GP1:
	UF : 7, UT : 3,	CONFIG : 'F U T, 0, 0, 0',
	X =   380.163  mm,	Y =     0.000  mm,	Z =     0.000  mm,
	W =  -167.364 deg,	P =     0.000 deg,	R =   105.687 deg
};
P[295]{
   GP1:
	UF : 7, UT : 3,	CONFIG : 'F U T, 0, 0, 0',
	X =   380.163  mm,	Y =     0.000  mm,	Z =     0.000  mm,
	W =  -167.364 deg,	P =     0.000 deg,	R =   105.687 deg
};
P[296]{
   GP1:
	UF : 7, UT : 3,	CONFIG : 'F U T, 0, 0, 0',
	X =   380.163  mm,	Y =     0.000  mm,	Z =     0.000  mm,
	W =  -167.364 deg,	P =     0.000 deg,	R =   105.687 deg
};
P[297]{
   GP1:
	UF : 7, UT : 3,	CONFIG : 'F U T, 0, 0, 0',
	X =   377.029  mm,	Y =     0.000  mm,	Z =     0.000  mm,
	W =  -167.364 deg,	P =     0.000 deg,	R =   105.687 deg
};
P[298]{
   GP1:
	UF : 7, UT : 3,	CONFIG : 'F U T, 0, 0, 0',
	X =   377.029  mm,	Y =     0.000  mm,	Z =     0.000  mm,
	W =  -167.364 deg,	P =     0.000 deg,	R =   105.687 deg
};
P[299]{
   GP1:
	UF : 7, UT : 3,	CONFIG : 'F U T, 0, 0, 0',
	X =   377.029  mm,	Y =     0.000  mm,	Z =     0.000  mm,
	W =  -167.364 deg,	P =     0.000 deg,	R =   105.687 deg
};
P[300]{
   GP1:
	UF : 7, UT : 3,	CONFIG : 'F U T, 0, 0, 0',
	X =   377.029  mm,	Y =     0.000  mm,	Z =     0.000  mm,
	W =  -167.364 deg,	P =     0.000 deg,	R =   105.687 deg
};
P[301]{
   GP1:
	UF : 7, UT : 3,	CONFIG : 'F U T, 0, 0, 0',
	X =   375.961  mm,	Y =    28.078  mm,	Z =     0.000  mm,
	W =  -167.364 deg,	P =    -0.001 deg,	R =   109.383 deg
};
P[302]{
   GP1:
	UF : 7, UT : 3,	CONFIG : 'F U T, 0, 0, 0',
	X =   373.304  mm,	Y =    52.730  mm,	Z =     0.000  mm,
	W =  -167.364 deg,	P =    -0.001 deg,	R =   113.116 deg
};
P[303]{
   GP1:
	UF : 7, UT : 3,	CONFIG : 'F U T, 0, 0, 0',
	X =   369.096  mm,	Y =    76.862  mm,	Z =     0.000  mm,
	W =  -167.364 deg,	P =    -0.001 deg,	R =   116.853 deg
};
P[304]{
   GP1:
	UF : 7, UT : 3,	CONFIG : 'F U T, 0, 0, 0',
	X =   363.362  mm,	Y =   100.533  mm,	Z =     0.000  mm,
	W =  -167.364 deg,	P =    -0.001 deg,	R =   120.597 deg
};
P[305]{
   GP1:
	UF : 7, UT : 3,	CONFIG : 'F U T, 0, 0, 0',
	X =   356.036  mm,	Y =   124.009  mm,	Z =     0.000  mm,
	W =  -167.364 deg,	P =    -0.001 deg,	R =   124.336 deg
};
P[306]{
   GP1:
	UF : 7, UT : 3,	CONFIG : 'F U T, 0, 0, 0',
	X =   347.130  mm,	Y =   147.117  mm,	Z =     0.000  mm,
	W =  -167.364 deg,	P =    -0.001 deg,	R =   128.067 deg
};
P[307]{
   GP1:
	UF : 7, UT : 3,	CONFIG : 'F U T, 0, 0, 0',
	X =   336.772  mm,	Y =   169.498  mm,	Z =     0.000  mm,
	W =  -167.364 deg,	P =    -0.001 deg,	R =   131.787 deg
};
P[308]{
   GP1:
	UF : 7, UT : 3,	CONFIG : 'F U T, 0, 0, 0',
	X =   325.018  mm,	Y =   191.073  mm,	Z =     0.000  mm,
	W =  -167.365 deg,	P =    -0.001 deg,	R =   135.514 deg
};
P[309]{
   GP1:
	UF : 7, UT : 3,	CONFIG : 'F U T, 0, 0, 0',
	X =   311.837  mm,	Y =   211.896  mm,	Z =     0.000  mm,
	W =  -167.365 deg,	P =    -0.001 deg,	R =   139.243 deg
};
P[310]{
   GP1:
	UF : 7, UT : 3,	CONFIG : 'F U T, 0, 0, 0',
	X =   297.346  mm,	Y =   231.791  mm,	Z =     0.000  mm,
	W =  -167.365 deg,	P =    -0.001 deg,	R =   142.946 deg
};
P[311]{
   GP1:
	UF : 7, UT : 3,	CONFIG : 'F U T, 0, 0, 0',
	X =   281.425  mm,	Y =   250.881  mm,	Z =     0.000  mm,
	W =  -167.365 deg,	P =    -0.001 deg,	R =   146.732 deg
};
P[312]{
   GP1:
	UF : 7, UT : 3,	CONFIG : 'F U T, 0, 0, 0',
	X =   264.507  mm,	Y =   268.664  mm,	Z =     0.000  mm,
	W =  -167.365 deg,	P =    -0.001 deg,	R =   150.457 deg
};
P[313]{
   GP1:
	UF : 7, UT : 3,	CONFIG : 'F U T, 0, 0, 0',
	X =   246.531  mm,	Y =   285.242  mm,	Z =     0.000  mm,
	W =  -167.366 deg,	P =    -0.001 deg,	R =   154.189 deg
};
P[314]{
   GP1:
	UF : 7, UT : 3,	CONFIG : 'F U T, 0, 0, 0',
	X =   227.419  mm,	Y =   300.695  mm,	Z =     0.000  mm,
	W =  -167.366 deg,	P =    -0.001 deg,	R =   157.904 deg
};
P[315]{
   GP1:
	UF : 7, UT : 3,	CONFIG : 'F U T, 0, 0, 0',
	X =   207.340  mm,	Y =   314.874  mm,	Z =     0.000  mm,
	W =  -167.366 deg,	P =    -0.001 deg,	R =   161.618 deg
};
P[316]{
   GP1:
	UF : 7, UT : 3,	CONFIG : 'F U T, 0, 0, 0',
	X =   186.516  mm,	Y =   327.639  mm,	Z =     0.000  mm,
	W =  -167.366 deg,	P =    -0.001 deg,	R =   165.350 deg
};
P[317]{
   GP1:
	UF : 7, UT : 3,	CONFIG : 'F U T, 0, 0, 0',
	X =   165.112  mm,	Y =   338.928  mm,	Z =     0.000  mm,
	W =  -167.366 deg,	P =    -0.001 deg,	R =   169.133 deg
};
P[318]{
   GP1:
	UF : 7, UT : 3,	CONFIG : 'F U T, 0, 0, 0',
	X =   142.609  mm,	Y =   348.993  mm,	Z =     0.000  mm,
	W =  -167.366 deg,	P =     0.000 deg,	R =   172.853 deg
};
P[319]{
   GP1:
	UF : 7, UT : 3,	CONFIG : 'F U T, 0, 0, 0',
	X =   119.501  mm,	Y =   357.567  mm,	Z =     0.000  mm,
	W =  -167.367 deg,	P =     0.000 deg,	R =   176.570 deg
};
P[320]{
   GP1:
	UF : 7, UT : 3,	CONFIG : 'F U T, 0, 0, 0',
	X =    95.904  mm,	Y =   364.607  mm,	Z =     0.000  mm,
	W =  -167.367 deg,	P =     0.000 deg,	R =  -179.686 deg
};
P[321]{
   GP1:
	UF : 7, UT : 3,	CONFIG : 'F U T, 0, 0, 0',
	X =    72.068  mm,	Y =   370.059  mm,	Z =     0.000  mm,
	W =  -167.367 deg,	P =     0.000 deg,	R =  -175.908 deg
};
P[322]{
   GP1:
	UF : 7, UT : 3,	CONFIG : 'F U T, 0, 0, 0',
	X =    47.917  mm,	Y =   373.954  mm,	Z =     0.000  mm,
	W =  -167.367 deg,	P =     0.000 deg,	R =  -172.154 deg
};
P[323]{
   GP1:
	UF : 7, UT : 3,	CONFIG : 'F U T, 0, 0, 0',
	X =    23.320  mm,	Y =   376.291  mm,	Z =     0.000  mm,
	W =  -167.367 deg,	P =     0.001 deg,	R =  -168.434 deg
};
P[324]{
   GP1:
	UF : 7, UT : 3,	CONFIG : 'F U T, 0, 0, 0',
	X =    -1.287  mm,	Y =   377.020  mm,	Z =     0.000  mm,
	W =  -167.367 deg,	P =     0.001 deg,	R =  -164.694 deg
};
P[325]{
   GP1:
	UF : 7, UT : 3,	CONFIG : 'F U T, 0, 0, 0',
	X =   -25.997  mm,	Y =   376.124  mm,	Z =     0.000  mm,
	W =  -167.367 deg,	P =     0.001 deg,	R =  -160.963 deg
};
P[326]{
   GP1:
	UF : 7, UT : 3,	CONFIG : 'F U T, 0, 0, 0',
	X =   -50.516  mm,	Y =   373.620  mm,	Z =     0.000  mm,
	W =  -167.367 deg,	P =     0.002 deg,	R =  -157.217 deg
};
P[327]{
   GP1:
	UF : 7, UT : 3,	CONFIG : 'F U T, 0, 0, 0',
	X =   -74.796  mm,	Y =   369.522  mm,	Z =     0.000  mm,
	W =  -167.367 deg,	P =     0.002 deg,	R =  -153.490 deg
};
P[328]{
   GP1:
	UF : 7, UT : 3,	CONFIG : 'F U T, 0, 0, 0',
	X =   -98.795  mm,	Y =   363.842  mm,	Z =     0.000  mm,
	W =  -167.367 deg,	P =     0.002 deg,	R =  -149.761 deg
};
P[329]{
   GP1:
	UF : 7, UT : 3,	CONFIG : 'F U T, 0, 0, 0',
	X =  -122.353  mm,	Y =   356.616  mm,	Z =     0.000  mm,
	W =  -167.367 deg,	P =     0.003 deg,	R =  -146.032 deg
};
P[330]{
   GP1:
	UF : 7, UT : 3,	CONFIG : 'F U T, 0, 0, 0',
	X =  -145.343  mm,	Y =   347.880  mm,	Z =     0.001  mm,
	W =  -167.367 deg,	P =     0.003 deg,	R =  -142.300 deg
};
P[331]{
   GP1:
	UF : 7, UT : 3,	CONFIG : 'F U T, 0, 0, 0',
	X =  -167.770  mm,	Y =   337.634  mm,	Z =     0.001  mm,
	W =  -167.367 deg,	P =     0.003 deg,	R =  -138.573 deg
};
P[332]{
   GP1:
	UF : 7, UT : 3,	CONFIG : 'F U T, 0, 0, 0',
	X =  -189.499  mm,	Y =   325.929  mm,	Z =     0.002  mm,
	W =  -167.367 deg,	P =     0.003 deg,	R =  -134.841 deg
};
P[333]{
   GP1:
	UF : 7, UT : 3,	CONFIG : 'F U T, 0, 0, 0',
	X =  -210.445  mm,	Y =   312.810  mm,	Z =     0.005  mm,
	W =  -167.367 deg,	P =     0.004 deg,	R =  -131.105 deg
};
P[334]{
   GP1:
	UF : 7, UT : 3,	CONFIG : 'F U T, 0, 0, 0',
	X =  -230.276  mm,	Y =   298.515  mm,	Z =     0.010  mm,
	W =  -167.367 deg,	P =     0.004 deg,	R =  -127.344 deg
};
P[335]{
   GP1:
	UF : 7, UT : 3,	CONFIG : 'F U T, 0, 0, 0',
	X =  -249.094  mm,	Y =   282.999  mm,	Z =     0.016  mm,
	W =  -167.366 deg,	P =     0.004 deg,	R =  -123.591 deg
};
P[336]{
   GP1:
	UF : 7, UT : 3,	CONFIG : 'F U T, 0, 0, 0',
	X =  -267.055  mm,	Y =   266.113  mm,	Z =     0.022  mm,
	W =  -167.366 deg,	P =     0.005 deg,	R =  -119.862 deg
};
P[337]{
   GP1:
	UF : 7, UT : 3,	CONFIG : 'F U T, 0, 0, 0',
	X =  -284.060  mm,	Y =   247.878  mm,	Z =     0.026  mm,
	W =  -167.366 deg,	P =     0.005 deg,	R =  -116.167 deg
};
P[338]{
   GP1:
	UF : 7, UT : 3,	CONFIG : 'F U T, 0, 0, 0',
	X =  -299.641  mm,	Y =   228.799  mm,	Z =     0.046  mm,
	W =  -167.366 deg,	P =     0.005 deg,	R =  -112.395 deg
};
P[339]{
   GP1:
	UF : 7, UT : 3,	CONFIG : 'F U T, 0, 0, 0',
	X =  -313.702  mm,	Y =   209.108  mm,	Z =     0.134  mm,
	W =  -167.365 deg,	P =     0.006 deg,	R =  -108.621 deg
};
P[340]{
   GP1:
	UF : 7, UT : 3,	CONFIG : 'F U T, 0, 0, 0',
	X =  -326.382  mm,	Y =   188.719  mm,	Z =     0.436  mm,
	W =  -167.365 deg,	P =     0.006 deg,	R =  -104.905 deg
};
P[341]{
   GP1:
	UF : 7, UT : 3,	CONFIG : 'F U T, 0, 0, 0',
	X =  -337.658  mm,	Y =   167.791  mm,	Z =     0.969  mm,
	W =  -167.365 deg,	P =     0.006 deg,	R =  -101.351 deg
};
P[342]{
   GP1:
	UF : 7, UT : 3,	CONFIG : 'F U T, 0, 0, 0',
	X =  -347.254  mm,	Y =   146.872  mm,	Z =     0.779  mm,
	W =  -167.364 deg,	P =     0.006 deg,	R =   -97.858 deg
};
P[343]{
   GP1:
	UF : 7, UT : 3,	CONFIG : 'F U T, 0, 0, 0',
	X =  -356.115  mm,	Y =   123.795  mm,	Z =     0.347  mm,
	W =  -167.364 deg,	P =     0.006 deg,	R =   -94.142 deg
};
P[344]{
   GP1:
	UF : 7, UT : 3,	CONFIG : 'F U T, 0, 0, 0',
	X =  -363.392  mm,	Y =   100.425  mm,	Z =     0.069  mm,
	W =  -167.364 deg,	P =     0.007 deg,	R =   -90.467 deg
};
P[345]{
   GP1:
	UF : 7, UT : 3,	CONFIG : 'F U T, 0, 0, 0',
	X =  -369.119  mm,	Y =    76.750  mm,	Z =     0.016  mm,
	W =  -167.363 deg,	P =     0.007 deg,	R =   -86.722 deg
};
P[346]{
   GP1:
	UF : 7, UT : 3,	CONFIG : 'F U T, 0, 1, 0',
	X =  -373.319  mm,	Y =    52.632  mm,	Z =     0.007  mm,
	W =  -167.363 deg,	P =     0.007 deg,	R =   -82.995 deg
};
P[347]{
   GP1:
	UF : 7, UT : 3,	CONFIG : 'F U T, 0, 1, 0',
	X =  -375.964  mm,	Y =    28.036  mm,	Z =     0.004  mm,
	W =  -167.362 deg,	P =     0.007 deg,	R =   -79.279 deg
};
P[348]{
   GP1:
	UF : 7, UT : 3,	CONFIG : 'F U T, 0, 1, 0',
	X =  -377.029  mm,	Y =     0.000  mm,	Z =     0.000  mm,
	W =  -167.362 deg,	P =     0.007 deg,	R =   -75.580 deg
};
P[349]{
   GP1:
	UF : 7, UT : 3,	CONFIG : 'F U T, 0, 1, 0',
	X =  -377.029  mm,	Y =     0.000  mm,	Z =     0.000  mm,
	W =  -167.362 deg,	P =     0.007 deg,	R =   -75.580 deg
};
P[350]{
   GP1:
	UF : 7, UT : 3,	CONFIG : 'F U T, 0, 1, 0',
	X =  -377.029  mm,	Y =     0.000  mm,	Z =     0.000  mm,
	W =  -167.362 deg,	P =     0.007 deg,	R =   -75.580 deg
};
P[351]{
   GP1:
	UF : 7, UT : 3,	CONFIG : 'F U T, 0, 1, 0',
	X =  -377.029  mm,	Y =     0.000  mm,	Z =     0.000  mm,
	W =  -167.362 deg,	P =     0.007 deg,	R =   -75.580 deg
};
P[352]{
   GP1:
	UF : 7, UT : 3,	CONFIG : 'F U T, 0, 1, 0',
	X =  -373.895  mm,	Y =     0.000  mm,	Z =     0.000  mm,
	W =  -167.361 deg,	P =     0.008 deg,	R =   -75.580 deg
};
P[353]{
   GP1:
	UF : 7, UT : 3,	CONFIG : 'F U T, 0, 1, 0',
	X =  -373.895  mm,	Y =     0.000  mm,	Z =     0.000  mm,
	W =  -167.361 deg,	P =     0.008 deg,	R =   -75.580 deg
};
P[354]{
   GP1:
	UF : 7, UT : 3,	CONFIG : 'F U T, 0, 1, 0',
	X =  -373.895  mm,	Y =     0.000  mm,	Z =     0.000  mm,
	W =  -167.361 deg,	P =     0.008 deg,	R =   -75.580 deg
};
P[355]{
   GP1:
	UF : 7, UT : 3,	CONFIG : 'F U T, 0, 1, 0',
	X =  -373.895  mm,	Y =     0.000  mm,	Z =     0.000  mm,
	W =  -167.361 deg,	P =     0.008 deg,	R =   -75.580 deg
};
P[356]{
   GP1:
	UF : 7, UT : 3,	CONFIG : 'F U T, 0, 1, 0',
	X =  -372.960  mm,	Y =    26.283  mm,	Z =     0.004  mm,
	W =  -167.368 deg,	P =     0.017 deg,	R =   -79.012 deg
};
P[357]{
   GP1:
	UF : 7, UT : 3,	CONFIG : 'F U T, 0, 1, 0',
	X =  -370.649  mm,	Y =    49.067  mm,	Z =     0.006  mm,
	W =  -167.374 deg,	P =     0.025 deg,	R =   -82.468 deg
};
P[358]{
   GP1:
	UF : 7, UT : 3,	CONFIG : 'F U T, 0, 0, 0',
	X =  -366.989  mm,	Y =    71.439  mm,	Z =     0.012  mm,
	W =  -167.381 deg,	P =     0.032 deg,	R =   -85.938 deg
};
P[359]{
   GP1:
	UF : 7, UT : 3,	CONFIG : 'F U T, 0, 0, 0',
	X =  -362.874  mm,	Y =    90.067  mm,	Z =     0.032  mm,
	W =  -167.401 deg,	P =     0.130 deg,	R =   -88.885 deg
};
P[360]{
   GP1:
	UF : 7, UT : 3,	CONFIG : 'F U T, 0, 0, 0',
	X =  -357.576  mm,	Y =   109.180  mm,	Z =     0.145  mm,
	W =  -167.280 deg,	P =     0.631 deg,	R =   -92.009 deg
};
P[361]{
   GP1:
	UF : 7, UT : 3,	CONFIG : 'F U T, 0, 0, 0',
	X =  -352.631  mm,	Y =   124.245  mm,	Z =     0.399  mm,
	W =  -166.740 deg,	P =     1.020 deg,	R =   -94.450 deg
};
P[362]{
   GP1:
	UF : 7, UT : 3,	CONFIG : 'F U T, 0, 0, 0',
	X =  -347.785  mm,	Y =   137.267  mm,	Z =     0.678  mm,
	W =  -166.135 deg,	P =     0.840 deg,	R =   -96.444 deg
};
P[363]{
   GP1:
	UF : 7, UT : 3,	CONFIG : 'F U T, 0, 0, 0',
	X =  -340.966  mm,	Y =   153.463  mm,	Z =     1.000  mm,
	W =  -165.835 deg,	P =     0.499 deg,	R =   -98.975 deg
};
P[364]{
   GP1:
	UF : 7, UT : 3,	CONFIG : 'F U T, 0, 0, 0',
	X =  -340.966  mm,	Y =   153.463  mm,	Z =     1.000  mm,
	W =  -165.835 deg,	P =     0.499 deg,	R =   -98.975 deg
};
P[365]{
   GP1:
	UF : 7, UT : 3,	CONFIG : 'F U T, 0, 0, 0',
	X =  -340.966  mm,	Y =   153.463  mm,	Z =     1.000  mm,
	W =  -165.835 deg,	P =     0.499 deg,	R =   -98.975 deg
};
P[366]{
   GP1:
	UF : 7, UT : 3,	CONFIG : 'F U T, 0, 0, 0',
	X =  -340.966  mm,	Y =   153.463  mm,	Z =     1.000  mm,
	W =  -165.835 deg,	P =     0.499 deg,	R =   -98.975 deg
};
P[367]{
   GP1:
	UF : 7, UT : 3,	CONFIG : 'F U T, 0, 0, 0',
	X =  -332.551  mm,	Y =   170.906  mm,	Z =     1.000  mm,
	W =  -165.925 deg,	P =    -1.651 deg,	R =  -101.891 deg
};
P[368]{
   GP1:
	UF : 7, UT : 3,	CONFIG : 'F U T, 0, 0, 0',
	X =  -332.551  mm,	Y =   170.906  mm,	Z =     1.000  mm,
	W =  -165.925 deg,	P =    -1.651 deg,	R =  -101.891 deg
};
P[369]{
   GP1:
	UF : 7, UT : 3,	CONFIG : 'F U T, 0, 0, 0',
	X =  -332.551  mm,	Y =   170.906  mm,	Z =     1.000  mm,
	W =  -165.925 deg,	P =    -1.651 deg,	R =  -101.891 deg
};
P[370]{
   GP1:
	UF : 7, UT : 3,	CONFIG : 'F U T, 0, 0, 0',
	X =  -332.551  mm,	Y =   170.906  mm,	Z =     1.000  mm,
	W =  -165.925 deg,	P =    -1.651 deg,	R =  -101.891 deg
};
P[371]{
   GP1:
	UF : 7, UT : 3,	CONFIG : 'F U T, 0, 0, 0',
	X =  -328.929  mm,	Y =   177.763  mm,	Z =     0.796  mm,
	W =  -166.242 deg,	P =    -2.045 deg,	R =  -103.389 deg
};
P[372]{
   GP1:
	UF : 7, UT : 3,	CONFIG : 'F U T, 0, 0, 0',
	X =  -326.909  mm,	Y =   181.475  mm,	Z =     0.668  mm,
	W =  -166.456 deg,	P =    -1.965 deg,	R =  -104.002 deg
};
P[373]{
   GP1:
	UF : 7, UT : 3,	CONFIG : 'F U T, 0, 0, 0',
	X =  -318.972  mm,	Y =   195.061  mm,	Z =     0.310  mm,
	W =  -167.126 deg,	P =    -1.028 deg,	R =  -106.371 deg
};
P[374]{
   GP1:
	UF : 7, UT : 3,	CONFIG : 'F U T, 0, 0, 0',
	X =  -314.162  mm,	Y =   202.710  mm,	Z =     0.192  mm,
	W =  -167.315 deg,	P =    -0.628 deg,	R =  -107.749 deg
};
P[375]{
   GP1:
	UF : 7, UT : 3,	CONFIG : 'F U T, 0, 0, 0',
	X =  -307.956  mm,	Y =   212.010  mm,	Z =     0.105  mm,
	W =  -167.415 deg,	P =    -0.317 deg,	R =  -109.567 deg
};
P[376]{
   GP1:
	UF : 7, UT : 3,	CONFIG : 'F U T, 0, 0, 0',
	X =  -299.660  mm,	Y =   223.588  mm,	Z =     0.053  mm,
	W =  -167.437 deg,	P =    -0.114 deg,	R =  -111.663 deg
};
P[377]{
   GP1:
	UF : 7, UT : 3,	CONFIG : 'F U T, 0, 0, 0',
	X =  -291.644  mm,	Y =   233.935  mm,	Z =     0.033  mm,
	W =  -167.411 deg,	P =    -0.061 deg,	R =  -113.645 deg
};
P[378]{
   GP1:
	UF : 7, UT : 3,	CONFIG : 'F U T, 0, 0, 0',
	X =  -283.505  mm,	Y =   243.745  mm,	Z =     0.027  mm,
	W =  -167.389 deg,	P =    -0.008 deg,	R =  -115.671 deg
};
P[379]{
   GP1:
	UF : 7, UT : 3,	CONFIG : 'F U T, 0, 0, 0',
	X =  -272.443  mm,	Y =   256.054  mm,	Z =     0.025  mm,
	W =  -167.374 deg,	P =    -0.014 deg,	R =  -118.208 deg
};
P[380]{
   GP1:
	UF : 7, UT : 3,	CONFIG : 'F U T, 0, 0, 0',
	X =  -260.885  mm,	Y =   267.826  mm,	Z =     0.022  mm,
	W =  -167.358 deg,	P =    -0.019 deg,	R =  -120.727 deg
};
P[381]{
   GP1:
	UF : 7, UT : 3,	CONFIG : 'F U T, 0, 0, 0',
	X =  -248.855  mm,	Y =   279.040  mm,	Z =     0.018  mm,
	W =  -167.342 deg,	P =    -0.022 deg,	R =  -123.242 deg
};
P[382]{
   GP1:
	UF : 7, UT : 3,	CONFIG : 'F U T, 0, 0, 0',
	X =  -231.547  mm,	Y =   293.551  mm,	Z =     0.012  mm,
	W =  -167.343 deg,	P =    -0.018 deg,	R =  -126.604 deg
};
P[383]{
   GP1:
	UF : 7, UT : 3,	CONFIG : 'F U T, 0, 0, 0',
	X =  -214.286  mm,	Y =   306.369  mm,	Z =     0.007  mm,
	W =  -167.345 deg,	P =    -0.015 deg,	R =  -130.089 deg
};
P[384]{
   GP1:
	UF : 7, UT : 3,	CONFIG : 'F U T, 0, 0, 0',
	X =  -195.447  mm,	Y =   318.736  mm,	Z =     0.003  mm,
	W =  -167.348 deg,	P =    -0.011 deg,	R =  -133.464 deg
};
P[385]{
   GP1:
	UF : 7, UT : 3,	CONFIG : 'F U T, 0, 0, 0',
	X =  -175.920  mm,	Y =   329.907  mm,	Z =     0.001  mm,
	W =  -167.350 deg,	P =    -0.008 deg,	R =  -136.824 deg
};
P[386]{
   GP1:
	UF : 7, UT : 3,	CONFIG : 'F U T, 0, 0, 0',
	X =  -156.361  mm,	Y =   339.605  mm,	Z =     0.001  mm,
	W =  -167.353 deg,	P =    -0.006 deg,	R =  -140.263 deg
};
P[387]{
   GP1:
	UF : 7, UT : 3,	CONFIG : 'F U T, 0, 0, 0',
	X =  -135.860  mm,	Y =   348.325  mm,	Z =     0.000  mm,
	W =  -167.356 deg,	P =    -0.003 deg,	R =  -143.682 deg
};
P[388]{
   GP1:
	UF : 7, UT : 3,	CONFIG : 'F U T, 0, 0, 0',
	X =  -114.694  mm,	Y =   355.856  mm,	Z =     0.000  mm,
	W =  -167.360 deg,	P =    -0.002 deg,	R =  -147.047 deg
};
P[389]{
   GP1:
	UF : 7, UT : 3,	CONFIG : 'F U T, 0, 0, 0',
	X =   -90.745  mm,	Y =   362.708  mm,	Z =     0.000  mm,
	W =  -167.364 deg,	P =     0.000 deg,	R =  -150.365 deg
};
P[390]{
   GP1:
	UF : 7, UT : 3,	CONFIG : 'F U T, 0, 0, 0',
	X =   -90.745  mm,	Y =   362.708  mm,	Z =     0.000  mm,
	W =  -167.364 deg,	P =     0.000 deg,	R =  -150.365 deg
};
P[391]{
   GP1:
	UF : 7, UT : 3,	CONFIG : 'F U T, 0, 0, 0',
	X =   -90.745  mm,	Y =   362.708  mm,	Z =     0.000  mm,
	W =  -167.364 deg,	P =     0.000 deg,	R =  -150.365 deg
};
P[392]{
   GP1:
	UF : 7, UT : 3,	CONFIG : 'F U T, 0, 0, 0',
	X =   -90.745  mm,	Y =   362.708  mm,	Z =     0.000  mm,
	W =  -167.364 deg,	P =     0.000 deg,	R =  -150.365 deg
};
P[393]{
   GP1:
	UF : 7, UT : 3,	CONFIG : 'F U T, 0, 0, 0',
	X =   -75.603  mm,	Y =   366.156  mm,	Z =     0.000  mm,
	W =  -167.364 deg,	P =     0.000 deg,	R =  -153.159 deg
};
P[394]{
   GP1:
	UF : 7, UT : 3,	CONFIG : 'F U T, 0, 0, 0',
	X =   -75.603  mm,	Y =   366.156  mm,	Z =     0.000  mm,
	W =  -167.364 deg,	P =     0.000 deg,	R =  -153.159 deg
};
P[395]{
   GP1:
	UF : 7, UT : 3,	CONFIG : 'F U T, 0, 0, 0',
	X =   -75.603  mm,	Y =   366.156  mm,	Z =     0.000  mm,
	W =  -167.364 deg,	P =     0.000 deg,	R =  -153.159 deg
};
P[396]{
   GP1:
	UF : 7, UT : 3,	CONFIG : 'F U T, 0, 0, 0',
	X =   -75.603  mm,	Y =   366.156  mm,	Z =     0.000  mm,
	W =  -167.364 deg,	P =     0.000 deg,	R =  -153.159 deg
};
P[397]{
   GP1:
	UF : 7, UT : 3,	CONFIG : 'F U T, 0, 0, 0',
	X =   -54.592  mm,	Y =   369.868  mm,	Z =     0.000  mm,
	W =  -167.364 deg,	P =     0.000 deg,	R =  -156.587 deg
};
P[398]{
   GP1:
	UF : 7, UT : 3,	CONFIG : 'F U T, 0, 0, 0',
	X =   -32.771  mm,	Y =   372.443  mm,	Z =     0.000  mm,
	W =  -167.364 deg,	P =     0.000 deg,	R =  -159.930 deg
};
P[399]{
   GP1:
	UF : 7, UT : 3,	CONFIG : 'F U T, 0, 0, 0',
	X =   -10.891  mm,	Y =   373.721  mm,	Z =     0.000  mm,
	W =  -167.364 deg,	P =     0.000 deg,	R =  -163.247 deg
};
P[400]{
   GP1:
	UF : 7, UT : 3,	CONFIG : 'F U T, 0, 0, 0',
	X =    10.990  mm,	Y =   373.717  mm,	Z =     0.000  mm,
	W =  -167.364 deg,	P =     0.000 deg,	R =  -166.651 deg
};
P[401]{
   GP1:
	UF : 7, UT : 3,	CONFIG : 'F U T, 0, 0, 0',
	X =    32.877  mm,	Y =   372.434  mm,	Z =     0.000  mm,
	W =  -167.364 deg,	P =     0.000 deg,	R =  -169.985 deg
};
P[402]{
   GP1:
	UF : 7, UT : 3,	CONFIG : 'F U T, 0, 0, 0',
	X =    54.635  mm,	Y =   369.862  mm,	Z =     0.000  mm,
	W =  -167.363 deg,	P =     0.000 deg,	R =  -173.305 deg
};
P[403]{
   GP1:
	UF : 7, UT : 3,	CONFIG : 'F U T, 0, 0, 0',
	X =    75.603  mm,	Y =   366.156  mm,	Z =     0.000  mm,
	W =  -167.363 deg,	P =     0.000 deg,	R =  -176.735 deg
};
P[404]{
   GP1:
	UF : 7, UT : 3,	CONFIG : 'F U T, 0, 0, 0',
	X =    75.603  mm,	Y =   366.156  mm,	Z =     0.000  mm,
	W =  -167.363 deg,	P =     0.000 deg,	R =  -176.735 deg
};
P[405]{
   GP1:
	UF : 7, UT : 3,	CONFIG : 'F U T, 0, 0, 0',
	X =    75.603  mm,	Y =   366.156  mm,	Z =     0.000  mm,
	W =  -167.363 deg,	P =     0.000 deg,	R =  -176.735 deg
};
P[406]{
   GP1:
	UF : 7, UT : 3,	CONFIG : 'F U T, 0, 0, 0',
	X =    75.603  mm,	Y =   366.156  mm,	Z =     0.000  mm,
	W =  -167.363 deg,	P =     0.000 deg,	R =  -176.735 deg
};
P[407]{
   GP1:
	UF : 7, UT : 3,	CONFIG : 'F U T, 0, 0, 0',
	X =    90.745  mm,	Y =   362.708  mm,	Z =     0.000  mm,
	W =  -167.363 deg,	P =     0.000 deg,	R =  -179.522 deg
};
P[408]{
   GP1:
	UF : 7, UT : 3,	CONFIG : 'F U T, 0, 0, 0',
	X =    90.745  mm,	Y =   362.708  mm,	Z =     0.000  mm,
	W =  -167.363 deg,	P =     0.000 deg,	R =  -179.522 deg
};
P[409]{
   GP1:
	UF : 7, UT : 3,	CONFIG : 'F U T, 0, 0, 0',
	X =    90.745  mm,	Y =   362.708  mm,	Z =     0.000  mm,
	W =  -167.363 deg,	P =     0.000 deg,	R =  -179.522 deg
};
P[410]{
   GP1:
	UF : 7, UT : 3,	CONFIG : 'F U T, 0, 0, 0',
	X =    90.745  mm,	Y =   362.708  mm,	Z =     0.000  mm,
	W =  -167.363 deg,	P =     0.000 deg,	R =  -179.522 deg
};
P[411]{
   GP1:
	UF : 7, UT : 3,	CONFIG : 'F U T, 0, 0, 0',
	X =   115.252  mm,	Y =   355.677  mm,	Z =     0.000  mm,
	W =  -167.363 deg,	P =     0.000 deg,	R =   177.058 deg
};
P[412]{
   GP1:
	UF : 7, UT : 3,	CONFIG : 'F U T, 0, 0, 0',
	X =   136.574  mm,	Y =   348.045  mm,	Z =     0.000  mm,
	W =  -167.364 deg,	P =     0.000 deg,	R =   173.657 deg
};
P[413]{
   GP1:
	UF : 7, UT : 3,	CONFIG : 'F U T, 0, 0, 0',
	X =   157.415  mm,	Y =   339.121  mm,	Z =     0.000  mm,
	W =  -167.364 deg,	P =     0.000 deg,	R =   170.180 deg
};
P[414]{
   GP1:
	UF : 7, UT : 3,	CONFIG : 'F U T, 0, 0, 0',
	X =   177.347  mm,	Y =   329.137  mm,	Z =     0.000  mm,
	W =  -167.364 deg,	P =     0.000 deg,	R =   166.714 deg
};
P[415]{
   GP1:
	UF : 7, UT : 3,	CONFIG : 'F U T, 0, 0, 0',
	X =   196.759  mm,	Y =   317.923  mm,	Z =     0.000  mm,
	W =  -167.364 deg,	P =     0.000 deg,	R =   163.262 deg
};
P[416]{
   GP1:
	UF : 7, UT : 3,	CONFIG : 'F U T, 0, 0, 0',
	X =   215.798  mm,	Y =   305.317  mm,	Z =     0.000  mm,
	W =  -167.364 deg,	P =     0.000 deg,	R =   159.875 deg
};
P[417]{
   GP1:
	UF : 7, UT : 3,	CONFIG : 'F U T, 0, 0, 0',
	X =   233.306  mm,	Y =   292.145  mm,	Z =     0.000  mm,
	W =  -167.364 deg,	P =     0.000 deg,	R =   156.353 deg
};
P[418]{
   GP1:
	UF : 7, UT : 3,	CONFIG : 'F U T, 0, 0, 0',
	X =   250.569  mm,	Y =   277.495  mm,	Z =     0.000  mm,
	W =  -167.364 deg,	P =     0.000 deg,	R =   152.936 deg
};
P[419]{
   GP1:
	UF : 7, UT : 3,	CONFIG : 'F U T, 0, 0, 0',
	X =   266.854  mm,	Y =   261.874  mm,	Z =     0.000  mm,
	W =  -167.364 deg,	P =     0.000 deg,	R =   149.534 deg
};
P[420]{
   GP1:
	UF : 7, UT : 3,	CONFIG : 'F U T, 0, 0, 0',
	X =   282.137  mm,	Y =   245.321  mm,	Z =     0.000  mm,
	W =  -167.364 deg,	P =     0.000 deg,	R =   146.094 deg
};
P[421]{
   GP1:
	UF : 7, UT : 3,	CONFIG : 'F U T, 0, 0, 0',
	X =   296.143  mm,	Y =   228.217  mm,	Z =     0.000  mm,
	W =  -167.364 deg,	P =     0.000 deg,	R =   142.589 deg
};
P[422]{
   GP1:
	UF : 7, UT : 3,	CONFIG : 'F U T, 0, 0, 0',
	X =   309.455  mm,	Y =   209.840  mm,	Z =     0.000  mm,
	W =  -167.364 deg,	P =     0.000 deg,	R =   139.169 deg
};
P[423]{
   GP1:
	UF : 7, UT : 3,	CONFIG : 'F U T, 0, 0, 0',
	X =   321.659  mm,	Y =   190.580  mm,	Z =     0.000  mm,
	W =  -167.364 deg,	P =     0.000 deg,	R =   135.771 deg
};
P[424]{
   GP1:
	UF : 7, UT : 3,	CONFIG : 'F U T, 0, 0, 0',
	X =   333.407  mm,	Y =   169.188  mm,	Z =     0.000  mm,
	W =  -167.364 deg,	P =     0.000 deg,	R =   132.300 deg
};
P[425]{
   GP1:
	UF : 7, UT : 3,	CONFIG : 'F U T, 0, 0, 0',
	X =   333.407  mm,	Y =   169.188  mm,	Z =     0.000  mm,
	W =  -167.364 deg,	P =     0.000 deg,	R =   132.300 deg
};
P[426]{
   GP1:
	UF : 7, UT : 3,	CONFIG : 'F U T, 0, 0, 0',
	X =   333.407  mm,	Y =   169.188  mm,	Z =     0.000  mm,
	W =  -167.364 deg,	P =     0.000 deg,	R =   132.300 deg
};
P[427]{
   GP1:
	UF : 7, UT : 3,	CONFIG : 'F U T, 0, 0, 0',
	X =   333.407  mm,	Y =   169.188  mm,	Z =     0.000  mm,
	W =  -167.364 deg,	P =     0.000 deg,	R =   132.300 deg
};
P[428]{
   GP1:
	UF : 7, UT : 3,	CONFIG : 'F U T, 0, 0, 0',
	X =   340.151  mm,	Y =   155.173  mm,	Z =     0.000  mm,
	W =  -167.364 deg,	P =     0.000 deg,	R =   130.208 deg
};
P[429]{
   GP1:
	UF : 7, UT : 3,	CONFIG : 'F U T, 0, 0, 0',
	X =   340.151  mm,	Y =   155.173  mm,	Z =     0.000  mm,
	W =  -167.364 deg,	P =     0.000 deg,	R =   130.208 deg
};
P[430]{
   GP1:
	UF : 7, UT : 3,	CONFIG : 'F U T, 0, 0, 0',
	X =   340.151  mm,	Y =   155.173  mm,	Z =     0.000  mm,
	W =  -167.364 deg,	P =     0.000 deg,	R =   130.208 deg
};
P[431]{
   GP1:
	UF : 7, UT : 3,	CONFIG : 'F U T, 0, 0, 0',
	X =   340.151  mm,	Y =   155.173  mm,	Z =     0.000  mm,
	W =  -167.364 deg,	P =     0.000 deg,	R =   130.208 deg
};
P[432]{
   GP1:
	UF : 7, UT : 3,	CONFIG : 'F U T, 0, 0, 0',
	X =   348.186  mm,	Y =   136.212  mm,	Z =     0.000  mm,
	W =  -167.364 deg,	P =     0.000 deg,	R =   126.375 deg
};
P[433]{
   GP1:
	UF : 7, UT : 3,	CONFIG : 'F U T, 0, 0, 0',
	X =   355.869  mm,	Y =   114.658  mm,	Z =     0.000  mm,
	W =  -167.364 deg,	P =     0.000 deg,	R =   122.950 deg
};
P[434]{
   GP1:
	UF : 7, UT : 3,	CONFIG : 'F U T, 0, 0, 0',
	X =   362.102  mm,	Y =    93.082  mm,	Z =     0.000  mm,
	W =  -167.364 deg,	P =     0.000 deg,	R =   119.465 deg
};
P[435]{
   GP1:
	UF : 7, UT : 3,	CONFIG : 'F U T, 0, 0, 0',
	X =   367.032  mm,	Y =    71.206  mm,	Z =     0.000  mm,
	W =  -167.364 deg,	P =     0.000 deg,	R =   115.966 deg
};
P[436]{
   GP1:
	UF : 7, UT : 3,	CONFIG : 'F U T, 0, 0, 0',
	X =   370.699  mm,	Y =    48.743  mm,	Z =     0.000  mm,
	W =  -167.364 deg,	P =     0.000 deg,	R =   112.514 deg
};
P[437]{
   GP1:
	UF : 7, UT : 3,	CONFIG : 'F U T, 0, 0, 0',
	X =   372.983  mm,	Y =    25.968  mm,	Z =     0.000  mm,
	W =  -167.364 deg,	P =     0.000 deg,	R =   109.100 deg
};
P[438]{
   GP1:
	UF : 7, UT : 3,	CONFIG : 'F U T, 0, 0, 0',
	X =   373.895  mm,	Y =     0.000  mm,	Z =     0.000  mm,
	W =  -167.364 deg,	P =     0.000 deg,	R =   105.687 deg
};
P[439]{
   GP1:
	UF : 7, UT : 3,	CONFIG : 'F U T, 0, 0, 0',
	X =   373.895  mm,	Y =     0.000  mm,	Z =     0.000  mm,
	W =  -167.364 deg,	P =     0.000 deg,	R =   105.687 deg
};
P[440]{
   GP1:
	UF : 7, UT : 3,	CONFIG : 'F U T, 0, 0, 0',
	X =   373.895  mm,	Y =     0.000  mm,	Z =     0.000  mm,
	W =  -167.364 deg,	P =     0.000 deg,	R =   105.687 deg
};
P[441]{
   GP1:
	UF : 7, UT : 3,	CONFIG : 'F U T, 0, 0, 0',
	X =   373.895  mm,	Y =     0.000  mm,	Z =     0.000  mm,
	W =  -167.364 deg,	P =     0.000 deg,	R =   105.687 deg
};
P[442]{
   GP1:
	UF : 7, UT : 3,	CONFIG : 'F U T, 0, 0, 0',
	X =   370.760  mm,	Y =     0.000  mm,	Z =     0.000  mm,
	W =  -167.364 deg,	P =    -0.001 deg,	R =   105.687 deg
};
P[443]{
   GP1:
	UF : 7, UT : 3,	CONFIG : 'F U T, 0, 0, 0',
	X =   370.760  mm,	Y =     0.000  mm,	Z =     0.000  mm,
	W =  -167.364 deg,	P =    -0.001 deg,	R =   105.687 deg
};
P[444]{
   GP1:
	UF : 7, UT : 3,	CONFIG : 'F U T, 0, 0, 0',
	X =   370.760  mm,	Y =     0.000  mm,	Z =     0.000  mm,
	W =  -167.364 deg,	P =    -0.001 deg,	R =   105.687 deg
};
P[445]{
   GP1:
	UF : 7, UT : 3,	CONFIG : 'F U T, 0, 0, 0',
	X =   370.760  mm,	Y =     0.000  mm,	Z =     0.000  mm,
	W =  -167.364 deg,	P =    -0.001 deg,	R =   105.687 deg
};
P[446]{
   GP1:
	UF : 7, UT : 3,	CONFIG : 'F U T, 0, 0, 0',
	X =   369.924  mm,	Y =    24.827  mm,	Z =     0.000  mm,
	W =  -167.364 deg,	P =     0.000 deg,	R =   108.903 deg
};
P[447]{
   GP1:
	UF : 7, UT : 3,	CONFIG : 'F U T, 0, 0, 0',
	X =   367.823  mm,	Y =    46.416  mm,	Z =     0.000  mm,
	W =  -167.364 deg,	P =     0.000 deg,	R =   112.119 deg
};
P[448]{
   GP1:
	UF : 7, UT : 3,	CONFIG : 'F U T, 0, 0, 0',
	X =   364.703  mm,	Y =    66.667  mm,	Z =     0.000  mm,
	W =  -167.364 deg,	P =     0.000 deg,	R =   115.488 deg
};
P[449]{
   GP1:
	UF : 7, UT : 3,	CONFIG : 'F U T, 0, 0, 0',
	X =   360.192  mm,	Y =    87.847  mm,	Z =     0.000  mm,
	W =  -167.364 deg,	P =     0.000 deg,	R =   118.720 deg
};
P[450]{
   GP1:
	UF : 7, UT : 3,	CONFIG : 'F U T, 0, 0, 0',
	X =   354.596  mm,	Y =   108.214  mm,	Z =     0.000  mm,
	W =  -167.364 deg,	P =     0.000 deg,	R =   122.021 deg
};
P[451]{
   GP1:
	UF : 7, UT : 3,	CONFIG : 'F U T, 0, 0, 0',
	X =   347.818  mm,	Y =   128.360  mm,	Z =     0.000  mm,
	W =  -167.364 deg,	P =     0.000 deg,	R =   125.301 deg
};
P[452]{
   GP1:
	UF : 7, UT : 3,	CONFIG : 'F U T, 0, 0, 0',
	X =   338.984  mm,	Y =   150.147  mm,	Z =     0.000  mm,
	W =  -167.364 deg,	P =     0.000 deg,	R =   128.494 deg
};
P[453]{
   GP1:
	UF : 7, UT : 3,	CONFIG : 'F U T, 0, 0, 0',
	X =   338.984  mm,	Y =   150.147  mm,	Z =     0.000  mm,
	W =  -167.364 deg,	P =     0.000 deg,	R =   128.494 deg
};
P[454]{
   GP1:
	UF : 7, UT : 3,	CONFIG : 'F U T, 0, 0, 0',
	X =   338.984  mm,	Y =   150.147  mm,	Z =     0.000  mm,
	W =  -167.364 deg,	P =     0.000 deg,	R =   128.494 deg
};
P[455]{
   GP1:
	UF : 7, UT : 3,	CONFIG : 'F U T, 0, 0, 0',
	X =   338.984  mm,	Y =   150.147  mm,	Z =     0.000  mm,
	W =  -167.364 deg,	P =     0.000 deg,	R =   128.494 deg
};
P[456]{
   GP1:
	UF : 7, UT : 3,	CONFIG : 'F U T, 0, 0, 0',
	X =   328.736  mm,	Y =   171.414  mm,	Z =     0.000  mm,
	W =  -167.364 deg,	P =     0.000 deg,	R =   132.163 deg
};
P[457]{
   GP1:
	UF : 7, UT : 3,	CONFIG : 'F U T, 0, 0, 0',
	X =   328.736  mm,	Y =   171.414  mm,	Z =     0.000  mm,
	W =  -167.364 deg,	P =     0.000 deg,	R =   132.163 deg
};
P[458]{
   GP1:
	UF : 7, UT : 3,	CONFIG : 'F U T, 0, 0, 0',
	X =   328.736  mm,	Y =   171.414  mm,	Z =     0.000  mm,
	W =  -167.364 deg,	P =     0.000 deg,	R =   132.163 deg
};
P[459]{
   GP1:
	UF : 7, UT : 3,	CONFIG : 'F U T, 0, 0, 0',
	X =   328.736  mm,	Y =   171.414  mm,	Z =     0.000  mm,
	W =  -167.364 deg,	P =     0.000 deg,	R =   132.163 deg
};
P[460]{
   GP1:
	UF : 7, UT : 3,	CONFIG : 'F U T, 0, 0, 0',
	X =   318.582  mm,	Y =   189.624  mm,	Z =     0.000  mm,
	W =  -167.364 deg,	P =     0.000 deg,	R =   135.876 deg
};
P[461]{
   GP1:
	UF : 7, UT : 3,	CONFIG : 'F U T, 0, 0, 0',
	X =   306.467  mm,	Y =   208.646  mm,	Z =     0.000  mm,
	W =  -167.364 deg,	P =     0.000 deg,	R =   139.312 deg
};
P[462]{
   GP1:
	UF : 7, UT : 3,	CONFIG : 'F U T, 0, 0, 0',
	X =   293.283  mm,	Y =   226.801  mm,	Z =     0.000  mm,
	W =  -167.364 deg,	P =     0.000 deg,	R =   142.716 deg
};
P[463]{
   GP1:
	UF : 7, UT : 3,	CONFIG : 'F U T, 0, 0, 0',
	X =   279.244  mm,	Y =   243.864  mm,	Z =     0.000  mm,
	W =  -167.364 deg,	P =     0.000 deg,	R =   146.181 deg
};
P[464]{
   GP1:
	UF : 7, UT : 3,	CONFIG : 'F U T, 0, 0, 0',
	X =   264.199  mm,	Y =   260.105  mm,	Z =     0.000  mm,
	W =  -167.364 deg,	P =     0.000 deg,	R =   149.659 deg
};
P[465]{
   GP1:
	UF : 7, UT : 3,	CONFIG : 'F U T, 0, 0, 0',
	X =   247.956  mm,	Y =   275.634  mm,	Z =     0.000  mm,
	W =  -167.364 deg,	P =     0.000 deg,	R =   153.036 deg
};
P[466]{
   GP1:
	UF : 7, UT : 3,	CONFIG : 'F U T, 0, 0, 0',
	X =   230.919  mm,	Y =   290.041  mm,	Z =     0.000  mm,
	W =  -167.364 deg,	P =     0.000 deg,	R =   156.491 deg
};
P[467]{
   GP1:
	UF : 7, UT : 3,	CONFIG : 'F U T, 0, 0, 0',
	X =   213.520  mm,	Y =   303.085  mm,	Z =     0.000  mm,
	W =  -167.364 deg,	P =     0.000 deg,	R =   159.986 deg
};
P[468]{
   GP1:
	UF : 7, UT : 3,	CONFIG : 'F U T, 0, 0, 0',
	X =   194.623  mm,	Y =   315.563  mm,	Z =     0.000  mm,
	W =  -167.364 deg,	P =     0.000 deg,	R =   163.392 deg
};
P[469]{
   GP1:
	UF : 7, UT : 3,	CONFIG : 'F U T, 0, 0, 0',
	X =   175.125  mm,	Y =   326.775  mm,	Z =     0.000  mm,
	W =  -167.364 deg,	P =     0.000 deg,	R =   166.803 deg
};
P[470]{
   GP1:
	UF : 7, UT : 3,	CONFIG : 'F U T, 0, 0, 0',
	X =   155.646  mm,	Y =   336.485  mm,	Z =     0.000  mm,
	W =  -167.364 deg,	P =     0.000 deg,	R =   170.301 deg
};
P[471]{
   GP1:
	UF : 7, UT : 3,	CONFIG : 'F U T, 0, 0, 0',
	X =   135.011  mm,	Y =   345.295  mm,	Z =     0.000  mm,
	W =  -167.364 deg,	P =     0.000 deg,	R =   173.722 deg
};
P[472]{
   GP1:
	UF : 7, UT : 3,	CONFIG : 'F U T, 0, 0, 0',
	X =   113.771  mm,	Y =   352.860  mm,	Z =     0.000  mm,
	W =  -167.363 deg,	P =     0.000 deg,	R =   177.138 deg
};
P[473]{
   GP1:
	UF : 7, UT : 3,	CONFIG : 'F U T, 0, 0, 0',
	X =    93.969  mm,	Y =   358.632  mm,	Z =     0.000  mm,
	W =  -167.363 deg,	P =     0.000 deg,	R =  -179.119 deg
};
P[474]{
   GP1:
	UF : 7, UT : 3,	CONFIG : 'F U T, 0, 0, 0',
	X =    93.969  mm,	Y =   358.632  mm,	Z =     0.000  mm,
	W =  -167.363 deg,	P =     0.000 deg,	R =  -179.119 deg
};
P[475]{
   GP1:
	UF : 7, UT : 3,	CONFIG : 'F U T, 0, 0, 0',
	X =    93.969  mm,	Y =   358.632  mm,	Z =     0.000  mm,
	W =  -167.363 deg,	P =     0.000 deg,	R =  -179.119 deg
};
P[476]{
   GP1:
	UF : 7, UT : 3,	CONFIG : 'F U T, 0, 0, 0',
	X =    93.969  mm,	Y =   358.632  mm,	Z =     0.000  mm,
	W =  -167.363 deg,	P =     0.000 deg,	R =  -179.119 deg
};
P[477]{
   GP1:
	UF : 7, UT : 3,	CONFIG : 'F U T, 0, 0, 0',
	X =    70.941  mm,	Y =   363.891  mm,	Z =     0.000  mm,
	W =  -167.363 deg,	P =     0.000 deg,	R =  -175.820 deg
};
P[478]{
   GP1:
	UF : 7, UT : 3,	CONFIG : 'F U T, 0, 0, 0',
	X =    70.941  mm,	Y =   363.891  mm,	Z =     0.000  mm,
	W =  -167.363 deg,	P =     0.000 deg,	R =  -175.820 deg
};
P[479]{
   GP1:
	UF : 7, UT : 3,	CONFIG : 'F U T, 0, 0, 0',
	X =    70.941  mm,	Y =   363.891  mm,	Z =     0.000  mm,
	W =  -167.363 deg,	P =     0.000 deg,	R =  -175.820 deg
};
P[480]{
   GP1:
	UF : 7, UT : 3,	CONFIG : 'F U T, 0, 0, 0',
	X =    70.941  mm,	Y =   363.891  mm,	Z =     0.000  mm,
	W =  -167.363 deg,	P =     0.000 deg,	R =  -175.820 deg
};
P[481]{
   GP1:
	UF : 7, UT : 3,	CONFIG : 'F U T, 0, 0, 0',
	X =    47.390  mm,	Y =   367.704  mm,	Z =     0.000  mm,
	W =  -167.363 deg,	P =     0.000 deg,	R =  -172.197 deg
};
P[482]{
   GP1:
	UF : 7, UT : 3,	CONFIG : 'F U T, 0, 0, 0',
	X =    23.724  mm,	Y =   369.992  mm,	Z =     0.000  mm,
	W =  -167.364 deg,	P =     0.000 deg,	R =  -168.579 deg
};
P[483]{
   GP1:
	UF : 7, UT : 3,	CONFIG : 'F U T, 0, 0, 0',
	X =    -0.137  mm,	Y =   370.760  mm,	Z =     0.000  mm,
	W =  -167.364 deg,	P =     0.000 deg,	R =  -164.919 deg
};
P[484]{
   GP1:
	UF : 7, UT : 3,	CONFIG : 'F U T, 0, 0, 0',
	X =   -23.919  mm,	Y =   369.980  mm,	Z =     0.000  mm,
	W =  -167.364 deg,	P =     0.000 deg,	R =  -161.273 deg
};
P[485]{
   GP1:
	UF : 7, UT : 3,	CONFIG : 'F U T, 0, 0, 0',
	X =   -47.470  mm,	Y =   367.693  mm,	Z =     0.000  mm,
	W =  -167.364 deg,	P =     0.000 deg,	R =  -157.654 deg
};
P[486]{
   GP1:
	UF : 7, UT : 3,	CONFIG : 'F U T, 0, 0, 0',
	X =   -70.941  mm,	Y =   363.891  mm,	Z =     0.000  mm,
	W =  -167.364 deg,	P =     0.000 deg,	R =  -154.058 deg
};
P[487]{
   GP1:
	UF : 7, UT : 3,	CONFIG : 'F U T, 0, 0, 0',
	X =   -70.941  mm,	Y =   363.891  mm,	Z =     0.000  mm,
	W =  -167.364 deg,	P =     0.000 deg,	R =  -154.058 deg
};
P[488]{
   GP1:
	UF : 7, UT : 3,	CONFIG : 'F U T, 0, 0, 0',
	X =   -70.941  mm,	Y =   363.891  mm,	Z =     0.000  mm,
	W =  -167.364 deg,	P =     0.000 deg,	R =  -154.058 deg
};
P[489]{
   GP1:
	UF : 7, UT : 3,	CONFIG : 'F U T, 0, 0, 0',
	X =   -70.941  mm,	Y =   363.891  mm,	Z =     0.000  mm,
	W =  -167.364 deg,	P =     0.000 deg,	R =  -154.058 deg
};
P[490]{
   GP1:
	UF : 7, UT : 3,	CONFIG : 'F U T, 0, 0, 0',
	X =   -93.969  mm,	Y =   358.632  mm,	Z =     0.000  mm,
	W =  -167.364 deg,	P =     0.000 deg,	R =  -150.900 deg
};
P[491]{
   GP1:
	UF : 7, UT : 3,	CONFIG : 'F U T, 0, 0, 0',
	X =   -93.969  mm,	Y =   358.632  mm,	Z =     0.000  mm,
	W =  -167.364 deg,	P =     0.000 deg,	R =  -150.900 deg
};
P[492]{
   GP1:
	UF : 7, UT : 3,	CONFIG : 'F U T, 0, 0, 0',
	X =   -93.969  mm,	Y =   358.632  mm,	Z =     0.000  mm,
	W =  -167.364 deg,	P =     0.000 deg,	R =  -150.900 deg
};
P[493]{
   GP1:
	UF : 7, UT : 3,	CONFIG : 'F U T, 0, 0, 0',
	X =   -93.969  mm,	Y =   358.632  mm,	Z =     0.000  mm,
	W =  -167.364 deg,	P =     0.000 deg,	R =  -150.900 deg
};
P[494]{
   GP1:
	UF : 7, UT : 3,	CONFIG : 'F U T, 0, 0, 0',
	X =  -115.416  mm,	Y =   352.319  mm,	Z =     0.000  mm,
	W =  -167.361 deg,	P =    -0.002 deg,	R =  -146.725 deg
};
P[495]{
   GP1:
	UF : 7, UT : 3,	CONFIG : 'F U T, 0, 0, 0',
	X =  -138.187  mm,	Y =   344.026  mm,	Z =     0.001  mm,
	W =  -167.358 deg,	P =    -0.005 deg,	R =  -142.968 deg
};
P[496]{
   GP1:
	UF : 7, UT : 3,	CONFIG : 'F U T, 0, 0, 0',
	X =  -160.523  mm,	Y =   334.192  mm,	Z =     0.001  mm,
	W =  -167.356 deg,	P =    -0.007 deg,	R =  -139.234 deg
};
P[497]{
   GP1:
	UF : 7, UT : 3,	CONFIG : 'F U T, 0, 0, 0',
	X =  -182.131  mm,	Y =   322.931  mm,	Z =     0.002  mm,
	W =  -167.353 deg,	P =    -0.011 deg,	R =  -135.481 deg
};
P[498]{
   GP1:
	UF : 7, UT : 3,	CONFIG : 'F U T, 0, 0, 0',
	X =  -202.844  mm,	Y =   310.339  mm,	Z =     0.005  mm,
	W =  -167.352 deg,	P =    -0.014 deg,	R =  -131.729 deg
};
P[499]{
   GP1:
	UF : 7, UT : 3,	CONFIG : 'F U T, 0, 0, 0',
	X =  -222.707  mm,	Y =   296.403  mm,	Z =     0.010  mm,
	W =  -167.350 deg,	P =    -0.018 deg,	R =  -127.971 deg
};
P[500]{
   GP1:
	UF : 7, UT : 3,	CONFIG : 'F U T, 0, 0, 0',
	X =  -241.642  mm,	Y =   281.181  mm,	Z =     0.017  mm,
	W =  -167.350 deg,	P =    -0.022 deg,	R =  -124.238 deg
};
P[501]{
   GP1:
	UF : 7, UT : 3,	CONFIG : 'F U T, 0, 0, 0',
	X =  -253.690  mm,	Y =   270.361  mm,	Z =     0.022  mm,
	W =  -167.366 deg,	P =    -0.013 deg,	R =  -121.744 deg
};
P[502]{
   GP1:
	UF : 7, UT : 3,	CONFIG : 'F U T, 0, 0, 0',
	X =  -265.260  mm,	Y =   259.026  mm,	Z =     0.024  mm,
	W =  -167.381 deg,	P =    -0.002 deg,	R =  -119.251 deg
};
P[503]{
   GP1:
	UF : 7, UT : 3,	CONFIG : 'F U T, 0, 0, 0',
	X =  -276.291  mm,	Y =   247.231  mm,	Z =     0.024  mm,
	W =  -167.395 deg,	P =     0.009 deg,	R =  -116.768 deg
};
P[504]{
   GP1:
	UF : 7, UT : 3,	CONFIG : 'F U T, 0, 0, 0',
	X =  -285.313  mm,	Y =   236.744  mm,	Z =     0.026  mm,
	W =  -167.436 deg,	P =    -0.027 deg,	R =  -114.666 deg
};
P[505]{
   GP1:
	UF : 7, UT : 3,	CONFIG : 'F U T, 0, 0, 0',
	X =  -293.728  mm,	Y =   226.216  mm,	Z =     0.038  mm,
	W =  -167.480 deg,	P =    -0.059 deg,	R =  -112.500 deg
};
P[506]{
   GP1:
	UF : 7, UT : 3,	CONFIG : 'F U T, 0, 0, 0',
	X =  -302.686  mm,	Y =   214.094  mm,	Z =     0.080  mm,
	W =  -167.510 deg,	P =    -0.227 deg,	R =  -110.160 deg
};
P[507]{
   GP1:
	UF : 7, UT : 3,	CONFIG : 'F U T, 0, 0, 0',
	X =  -313.870  mm,	Y =   197.318  mm,	Z =     0.258  mm,
	W =  -167.382 deg,	P =    -0.867 deg,	R =  -107.210 deg
};
P[508]{
   GP1:
	UF : 7, UT : 3,	CONFIG : 'F U T, 0, 0, 0',
	X =  -324.532  mm,	Y =   179.281  mm,	Z =     0.764  mm,
	W =  -166.712 deg,	P =    -2.094 deg,	R =  -103.852 deg
};
P[509]{
   GP1:
	UF : 7, UT : 3,	CONFIG : 'F U T, 0, 0, 0',
	X =  -328.143  mm,	Y =   172.612  mm,	Z =     1.000  mm,
	W =  -166.445 deg,	P =    -1.885 deg,	R =  -102.978 deg
};
P[510]{
   GP1:
	UF : 7, UT : 3,	CONFIG : 'F U T, 0, 0, 0',
	X =  -328.143  mm,	Y =   172.612  mm,	Z =     1.000  mm,
	W =  -166.445 deg,	P =    -1.885 deg,	R =  -102.978 deg
};
P[511]{
   GP1:
	UF : 7, UT : 3,	CONFIG : 'F U T, 0, 0, 0',
	X =  -328.143  mm,	Y =   172.612  mm,	Z =     1.000  mm,
	W =  -166.445 deg,	P =    -1.885 deg,	R =  -102.978 deg
};
P[512]{
   GP1:
	UF : 7, UT : 3,	CONFIG : 'F U T, 0, 0, 0',
	X =  -328.143  mm,	Y =   172.612  mm,	Z =     1.000  mm,
	W =  -166.445 deg,	P =    -1.885 deg,	R =  -102.978 deg
};
P[513]{
   GP1:
	UF : 7, UT : 3,	CONFIG : 'F U T, 0, 0, 0',
	X =  -339.541  mm,	Y =   148.918  mm,	Z =     1.000  mm,
	W =  -166.246 deg,	P =     0.761 deg,	R =   -98.511 deg
};
P[514]{
   GP1:
	UF : 7, UT : 3,	CONFIG : 'F U T, 0, 0, 0',
	X =  -339.541  mm,	Y =   148.918  mm,	Z =     1.000  mm,
	W =  -166.246 deg,	P =     0.761 deg,	R =   -98.511 deg
};
P[515]{
   GP1:
	UF : 7, UT : 3,	CONFIG : 'F U T, 0, 0, 0',
	X =  -339.541  mm,	Y =   148.918  mm,	Z =     1.000  mm,
	W =  -166.246 deg,	P =     0.761 deg,	R =   -98.511 deg
};
P[516]{
   GP1:
	UF : 7, UT : 3,	CONFIG : 'F U T, 0, 0, 0',
	X =  -339.541  mm,	Y =   148.918  mm,	Z =     1.000  mm,
	W =  -166.246 deg,	P =     0.761 deg,	R =   -98.511 deg
};
P[517]{
   GP1:
	UF : 7, UT : 3,	CONFIG : 'F U T, 0, 0, 0',
	X =  -346.064  mm,	Y =   133.023  mm,	Z =     0.652  mm,
	W =  -166.437 deg,	P =     1.067 deg,	R =   -95.925 deg
};
P[518]{
   GP1:
	UF : 7, UT : 3,	CONFIG : 'F U T, 0, 0, 0',
	X =  -349.900  mm,	Y =   122.576  mm,	Z =     0.396  mm,
	W =  -166.950 deg,	P =     1.202 deg,	R =   -94.278 deg
};
P[519]{
   GP1:
	UF : 7, UT : 3,	CONFIG : 'F U T, 0, 0, 0',
	X =  -354.794  mm,	Y =   107.569  mm,	Z =     0.128  mm,
	W =  -167.395 deg,	P =     0.655 deg,	R =   -91.881 deg
};
P[520]{
   GP1:
	UF : 7, UT : 3,	CONFIG : 'F U T, 0, 0, 0',
	X =  -359.787  mm,	Y =    89.495  mm,	Z =     0.028  mm,
	W =  -167.434 deg,	P =     0.129 deg,	R =   -88.920 deg
};
P[521]{
   GP1:
	UF : 7, UT : 3,	CONFIG : 'F U T, 0, 0, 0',
	X =  -364.010  mm,	Y =    70.316  mm,	Z =     0.010  mm,
	W =  -167.391 deg,	P =     0.027 deg,	R =   -85.797 deg
};
P[522]{
   GP1:
	UF : 7, UT : 3,	CONFIG : 'F U T, 0, 1, 0',
	X =  -367.616  mm,	Y =    48.091  mm,	Z =     0.006  mm,
	W =  -167.381 deg,	P =     0.022 deg,	R =   -82.356 deg
};
P[523]{
   GP1:
	UF : 7, UT : 3,	CONFIG : 'F U T, 0, 1, 0',
	X =  -369.861  mm,	Y =    25.673  mm,	Z =     0.004  mm,
	W =  -167.371 deg,	P =     0.016 deg,	R =   -78.957 deg
};
P[524]{
   GP1:
	UF : 7, UT : 3,	CONFIG : 'F U T, 0, 1, 0',
	X =  -370.760  mm,	Y =     0.000  mm,	Z =     0.000  mm,
	W =  -167.361 deg,	P =     0.008 deg,	R =   -75.582 deg
};
P[525]{
   GP1:
	UF : 7, UT : 3,	CONFIG : 'F U T, 0, 1, 0',
	X =  -370.760  mm,	Y =     0.000  mm,	Z =     0.000  mm,
	W =  -167.361 deg,	P =     0.008 deg,	R =   -75.582 deg
};
P[526]{
   GP1:
	UF : 7, UT : 3,	CONFIG : 'F U T, 0, 1, 0',
	X =  -370.760  mm,	Y =     0.000  mm,	Z =     0.000  mm,
	W =  -167.361 deg,	P =     0.008 deg,	R =   -75.582 deg
};
P[527]{
   GP1:
	UF : 7, UT : 3,	CONFIG : 'F U T, 0, 1, 0',
	X =  -370.760  mm,	Y =     0.000  mm,	Z =     0.000  mm,
	W =  -167.361 deg,	P =     0.008 deg,	R =   -75.582 deg
};
P[528]{
   GP1:
	UF : 7, UT : 3,	CONFIG : 'F U T, 0, 1, 0',
	X =  -367.626  mm,	Y =     0.000  mm,	Z =     0.000  mm,
	W =  -167.361 deg,	P =     0.009 deg,	R =   -75.583 deg
};
P[529]{
   GP1:
	UF : 7, UT : 3,	CONFIG : 'F U T, 0, 1, 0',
	X =  -367.626  mm,	Y =     0.000  mm,	Z =     0.000  mm,
	W =  -167.361 deg,	P =     0.009 deg,	R =   -75.583 deg
};
P[530]{
   GP1:
	UF : 7, UT : 3,	CONFIG : 'F U T, 0, 1, 0',
	X =  -367.626  mm,	Y =     0.000  mm,	Z =     0.000  mm,
	W =  -167.361 deg,	P =     0.009 deg,	R =   -75.583 deg
};
P[531]{
   GP1:
	UF : 7, UT : 3,	CONFIG : 'F U T, 0, 1, 0',
	X =  -367.626  mm,	Y =     0.000  mm,	Z =     0.000  mm,
	W =  -167.361 deg,	P =     0.009 deg,	R =   -75.583 deg
};
P[532]{
   GP1:
	UF : 7, UT : 3,	CONFIG : 'F U T, 0, 1, 0',
	X =  -366.712  mm,	Y =    25.767  mm,	Z =     0.004  mm,
	W =  -167.375 deg,	P =     0.016 deg,	R =   -78.999 deg
};
P[533]{
   GP1:
	UF : 7, UT : 3,	CONFIG : 'F U T, 0, 1, 0',
	X =  -364.422  mm,	Y =    48.337  mm,	Z =     0.006  mm,
	W =  -167.388 deg,	P =     0.020 deg,	R =   -82.487 deg
};
P[534]{
   GP1:
	UF : 7, UT : 3,	CONFIG : 'F U T, 0, 0, 0',
	X =  -360.757  mm,	Y =    70.661  mm,	Z =     0.008  mm,
	W =  -167.401 deg,	P =     0.023 deg,	R =   -85.987 deg
};
P[535]{
   GP1:
	UF : 7, UT : 3,	CONFIG : 'F U T, 0, 0, 0',
	X =  -356.466  mm,	Y =    89.851  mm,	Z =     0.023  mm,
	W =  -167.463 deg,	P =     0.130 deg,	R =   -89.137 deg
};
P[536]{
   GP1:
	UF : 7, UT : 3,	CONFIG : 'F U T, 0, 0, 0',
	X =  -353.958  mm,	Y =    99.240  mm,	Z =     0.054  mm,
	W =  -167.496 deg,	P =     0.340 deg,	R =   -90.679 deg
};
P[537]{
   GP1:
	UF : 7, UT : 3,	CONFIG : 'F U T, 0, 0, 0',
	X =  -348.872  mm,	Y =   115.854  mm,	Z =     0.261  mm,
	W =  -167.330 deg,	P =     1.146 deg,	R =   -93.261 deg
};
P[538]{
   GP1:
	UF : 7, UT : 3,	CONFIG : 'F U T, 0, 0, 0',
	X =  -344.938  mm,	Y =   127.131  mm,	Z =     0.548  mm,
	W =  -166.848 deg,	P =     1.437 deg,	R =   -95.127 deg
};
P[539]{
   GP1:
	UF : 7, UT : 3,	CONFIG : 'F U T, 0, 0, 0',
	X =  -340.607  mm,	Y =   138.315  mm,	Z =     0.840  mm,
	W =  -166.496 deg,	P =     1.054 deg,	R =   -97.009 deg
};
P[540]{
   GP1:
	UF : 7, UT : 3,	CONFIG : 'F U T, 0, 0, 0',
	X =  -337.521  mm,	Y =   145.693  mm,	Z =     1.000  mm,
	W =  -166.545 deg,	P =     0.895 deg,	R =   -98.904 deg
};
P[541]{
   GP1:
	UF : 7, UT : 3,	CONFIG : 'F U T, 0, 0, 0',
	X =  -337.521  mm,	Y =   145.693  mm,	Z =     1.000  mm,
	W =  -166.545 deg,	P =     0.895 deg,	R =   -98.904 deg
};
P[542]{
   GP1:
	UF : 7, UT : 3,	CONFIG : 'F U T, 0, 0, 0',
	X =  -337.521  mm,	Y =   145.693  mm,	Z =     1.000  mm,
	W =  -166.545 deg,	P =     0.895 deg,	R =   -98.904 deg
};
P[543]{
   GP1:
	UF : 7, UT : 3,	CONFIG : 'F U T, 0, 0, 0',
	X =  -337.521  mm,	Y =   145.693  mm,	Z =     1.000  mm,
	W =  -166.545 deg,	P =     0.895 deg,	R =   -98.904 deg
};
P[544]{
   GP1:
	UF : 7, UT : 3,	CONFIG : 'F U T, 0, 0, 0',
	X =  -324.360  mm,	Y =   173.046  mm,	Z =     1.000  mm,
	W =  -166.890 deg,	P =    -1.964 deg,	R =  -103.533 deg
};
P[545]{
   GP1:
	UF : 7, UT : 3,	CONFIG : 'F U T, 0, 0, 0',
	X =  -324.360  mm,	Y =   173.046  mm,	Z =     1.000  mm,
	W =  -166.890 deg,	P =    -1.964 deg,	R =  -103.533 deg
};
P[546]{
   GP1:
	UF : 7, UT : 3,	CONFIG : 'F U T, 0, 0, 0',
	X =  -324.360  mm,	Y =   173.046  mm,	Z =     1.000  mm,
	W =  -166.890 deg,	P =    -1.964 deg,	R =  -103.533 deg
};
P[547]{
   GP1:
	UF : 7, UT : 3,	CONFIG : 'F U T, 0, 0, 0',
	X =  -324.360  mm,	Y =   173.046  mm,	Z =     1.000  mm,
	W =  -166.890 deg,	P =    -1.964 deg,	R =  -103.533 deg
};
P[548]{
   GP1:
	UF : 7, UT : 3,	CONFIG : 'F U T, 0, 0, 0',
	X =  -320.775  mm,	Y =   179.595  mm,	Z =     0.748  mm,
	W =  -167.073 deg,	P =    -2.105 deg,	R =  -104.263 deg
};
P[549]{
   GP1:
	UF : 7, UT : 3,	CONFIG : 'F U T, 0, 0, 0',
	X =  -309.757  mm,	Y =   197.956  mm,	Z =     0.224  mm,
	W =  -167.556 deg,	P =    -0.783 deg,	R =  -107.423 deg
};
P[550]{
   GP1:
	UF : 7, UT : 3,	CONFIG : 'F U T, 0, 0, 0',
	X =  -298.424  mm,	Y =   214.673  mm,	Z =     0.061  mm,
	W =  -167.576 deg,	P =    -0.168 deg,	R =  -110.705 deg
};
P[551]{
   GP1:
	UF : 7, UT : 3,	CONFIG : 'F U T, 0, 0, 0',
	X =  -288.952  mm,	Y =   227.271  mm,	Z =     0.027  mm,
	W =  -167.506 deg,	P =    -0.020 deg,	R =  -113.167 deg
};
P[552]{
   GP1:
	UF : 7, UT : 3,	CONFIG : 'F U T, 0, 0, 0',
	X =  -280.075  mm,	Y =   238.116  mm,	Z =     0.021  mm,
	W =  -167.452 deg,	P =    -0.001 deg,	R =  -115.289 deg
};
P[553]{
   GP1:
	UF : 7, UT : 3,	CONFIG : 'F U T, 0, 0, 0',
	X =  -270.796  mm,	Y =   248.600  mm,	Z =     0.023  mm,
	W =  -167.400 deg,	P =     0.021 deg,	R =  -117.412 deg
};
P[554]{
   GP1:
	UF : 7, UT : 3,	CONFIG : 'F U T, 0, 0, 0',
	X =  -254.116  mm,	Y =   265.629  mm,	Z =     0.023  mm,
	W =  -167.379 deg,	P =    -0.002 deg,	R =  -121.228 deg
};
P[555]{
   GP1:
	UF : 7, UT : 3,	CONFIG : 'F U T, 0, 0, 0',
	X =  -236.204  mm,	Y =   281.674  mm,	Z =     0.017  mm,
	W =  -167.356 deg,	P =    -0.021 deg,	R =  -124.999 deg
};
P[556]{
   GP1:
	UF : 7, UT : 3,	CONFIG : 'F U T, 0, 0, 0',
	X =  -218.379  mm,	Y =   295.716  mm,	Z =     0.010  mm,
	W =  -167.356 deg,	P =    -0.018 deg,	R =  -128.571 deg
};
P[557]{
   GP1:
	UF : 7, UT : 3,	CONFIG : 'F U T, 0, 0, 0',
	X =  -199.558  mm,	Y =   308.743  mm,	Z =     0.005  mm,
	W =  -167.356 deg,	P =    -0.014 deg,	R =  -132.093 deg
};
P[558]{
   GP1:
	UF : 7, UT : 3,	CONFIG : 'F U T, 0, 0, 0',
	X =  -179.847  mm,	Y =   320.615  mm,	Z =     0.002  mm,
	W =  -167.357 deg,	P =    -0.011 deg,	R =  -135.621 deg
};
P[559]{
   GP1:
	UF : 7, UT : 3,	CONFIG : 'F U T, 0, 0, 0',
	X =  -159.799  mm,	Y =   331.060  mm,	Z =     0.001  mm,
	W =  -167.358 deg,	P =    -0.008 deg,	R =  -139.172 deg
};
P[560]{
   GP1:
	UF : 7, UT : 3,	CONFIG : 'F U T, 0, 0, 0',
	X =  -138.886  mm,	Y =   340.359  mm,	Z =     0.000  mm,
	W =  -167.360 deg,	P =    -0.005 deg,	R =  -142.709 deg
};
P[561]{
   GP1:
	UF : 7, UT : 3,	CONFIG : 'F U T, 0, 0, 0',
	X =  -117.896  mm,	Y =   348.192  mm,	Z =     0.000  mm,
	W =  -167.361 deg,	P =    -0.003 deg,	R =  -146.299 deg
};
P[562]{
   GP1:
	UF : 7, UT : 3,	CONFIG : 'F U T, 0, 0, 0',
	X =   -95.418  mm,	Y =   355.016  mm,	Z =     0.000  mm,
	W =  -167.364 deg,	P =     0.000 deg,	R =  -149.740 deg
};
P[563]{
   GP1:
	UF : 7, UT : 3,	CONFIG : 'F U T, 0, 0, 0',
	X =   -95.418  mm,	Y =   355.016  mm,	Z =     0.000  mm,
	W =  -167.364 deg,	P =     0.000 deg,	R =  -149.740 deg
};
P[564]{
   GP1:
	UF : 7, UT : 3,	CONFIG : 'F U T, 0, 0, 0',
	X =   -95.418  mm,	Y =   355.016  mm,	Z =     0.000  mm,
	W =  -167.364 deg,	P =     0.000 deg,	R =  -149.740 deg
};
P[565]{
   GP1:
	UF : 7, UT : 3,	CONFIG : 'F U T, 0, 0, 0',
	X =   -95.418  mm,	Y =   355.016  mm,	Z =     0.000  mm,
	W =  -167.364 deg,	P =     0.000 deg,	R =  -149.740 deg
};
P[566]{
   GP1:
	UF : 7, UT : 3,	CONFIG : 'F U T, 0, 0, 0',
	X =   -68.050  mm,	Y =   361.251  mm,	Z =     0.000  mm,
	W =  -167.363 deg,	P =     0.000 deg,	R =  -153.693 deg
};
P[567]{
   GP1:
	UF : 7, UT : 3,	CONFIG : 'F U T, 0, 0, 0',
	X =   -68.050  mm,	Y =   361.251  mm,	Z =     0.000  mm,
	W =  -167.363 deg,	P =     0.000 deg,	R =  -153.693 deg
};
P[568]{
   GP1:
	UF : 7, UT : 3,	CONFIG : 'F U T, 0, 0, 0',
	X =   -68.050  mm,	Y =   361.251  mm,	Z =     0.000  mm,
	W =  -167.363 deg,	P =     0.000 deg,	R =  -153.693 deg
};
P[569]{
   GP1:
	UF : 7, UT : 3,	CONFIG : 'F U T, 0, 0, 0',
	X =   -68.050  mm,	Y =   361.251  mm,	Z =     0.000  mm,
	W =  -167.363 deg,	P =     0.000 deg,	R =  -153.693 deg
};
P[570]{
   GP1:
	UF : 7, UT : 3,	CONFIG : 'F U T, 0, 0, 0',
	X =   -46.915  mm,	Y =   364.604  mm,	Z =     0.000  mm,
	W =  -167.364 deg,	P =     0.000 deg,	R =  -157.699 deg
};
P[571]{
   GP1:
	UF : 7, UT : 3,	CONFIG : 'F U T, 0, 0, 0',
	X =   -23.535  mm,	Y =   366.861  mm,	Z =     0.000  mm,
	W =  -167.364 deg,	P =     0.000 deg,	R =  -161.313 deg
};
P[572]{
   GP1:
	UF : 7, UT : 3,	CONFIG : 'F U T, 0, 0, 0',
	X =    -0.011  mm,	Y =   367.626  mm,	Z =     0.000  mm,
	W =  -167.363 deg,	P =     0.000 deg,	R =  -164.944 deg
};
P[573]{
   GP1:
	UF : 7, UT : 3,	CONFIG : 'F U T, 0, 0, 0',
	X =    23.544  mm,	Y =   366.861  mm,	Z =     0.000  mm,
	W =  -167.363 deg,	P =     0.000 deg,	R =  -168.582 deg
};
P[574]{
   GP1:
	UF : 7, UT : 3,	CONFIG : 'F U T, 0, 0, 0',
	X =    46.948  mm,	Y =   364.600  mm,	Z =     0.000  mm,
	W =  -167.363 deg,	P =     0.000 deg,	R =  -172.196 deg
};
P[575]{
   GP1:
	UF : 7, UT : 3,	CONFIG : 'F U T, 0, 0, 0',
	X =    68.050  mm,	Y =   361.251  mm,	Z =     0.000  mm,
	W =  -167.363 deg,	P =     0.000 deg,	R =  -176.214 deg
};
P[576]{
   GP1:
	UF : 7, UT : 3,	CONFIG : 'F U T, 0, 0, 0',
	X =    68.050  mm,	Y =   361.251  mm,	Z =     0.000  mm,
	W =  -167.363 deg,	P =     0.000 deg,	R =  -176.214 deg
};
P[577]{
   GP1:
	UF : 7, UT : 3,	CONFIG : 'F U T, 0, 0, 0',
	X =    68.050  mm,	Y =   361.251  mm,	Z =     0.000  mm,
	W =  -167.363 deg,	P =     0.000 deg,	R =  -176.214 deg
};
P[578]{
   GP1:
	UF : 7, UT : 3,	CONFIG : 'F U T, 0, 0, 0',
	X =    68.050  mm,	Y =   361.251  mm,	Z =     0.000  mm,
	W =  -167.363 deg,	P =     0.000 deg,	R =  -176.214 deg
};
P[579]{
   GP1:
	UF : 7, UT : 3,	CONFIG : 'F U T, 0, 0, 0',
	X =    95.418  mm,	Y =   355.016  mm,	Z =     0.000  mm,
	W =  -167.363 deg,	P =     0.000 deg,	R =   179.941 deg
};
P[580]{
   GP1:
	UF : 7, UT : 3,	CONFIG : 'F U T, 0, 0, 0',
	X =    95.418  mm,	Y =   355.016  mm,	Z =     0.000  mm,
	W =  -167.363 deg,	P =     0.000 deg,	R =   179.941 deg
};
P[581]{
   GP1:
	UF : 7, UT : 3,	CONFIG : 'F U T, 0, 0, 0',
	X =    95.418  mm,	Y =   355.016  mm,	Z =     0.000  mm,
	W =  -167.363 deg,	P =     0.000 deg,	R =   179.941 deg
};
P[582]{
   GP1:
	UF : 7, UT : 3,	CONFIG : 'F U T, 0, 0, 0',
	X =    95.418  mm,	Y =   355.016  mm,	Z =     0.000  mm,
	W =  -167.363 deg,	P =     0.000 deg,	R =   179.941 deg
};
P[583]{
   GP1:
	UF : 7, UT : 3,	CONFIG : 'F U T, 0, 0, 0',
	X =   116.379  mm,	Y =   348.696  mm,	Z =     0.000  mm,
	W =  -167.363 deg,	P =     0.000 deg,	R =   176.689 deg
};
P[584]{
   GP1:
	UF : 7, UT : 3,	CONFIG : 'F U T, 0, 0, 0',
	X =   135.984  mm,	Y =   341.536  mm,	Z =     0.000  mm,
	W =  -167.364 deg,	P =     0.000 deg,	R =   173.307 deg
};
P[585]{
   GP1:
	UF : 7, UT : 3,	CONFIG : 'F U T, 0, 0, 0',
	X =   155.790  mm,	Y =   332.968  mm,	Z =     0.000  mm,
	W =  -167.364 deg,	P =     0.000 deg,	R =   170.019 deg
};
P[586]{
   GP1:
	UF : 7, UT : 3,	CONFIG : 'F U T, 0, 0, 0',
	X =   174.347  mm,	Y =   323.632  mm,	Z =     0.000  mm,
	W =  -167.364 deg,	P =     0.000 deg,	R =   166.644 deg
};
P[587]{
   GP1:
	UF : 7, UT : 3,	CONFIG : 'F U T, 0, 0, 0',
	X =   193.093  mm,	Y =   312.825  mm,	Z =     0.000  mm,
	W =  -167.364 deg,	P =     0.000 deg,	R =   163.360 deg
};
P[588]{
   GP1:
	UF : 7, UT : 3,	CONFIG : 'F U T, 0, 0, 0',
	X =   211.069  mm,	Y =   300.973  mm,	Z =     0.000  mm,
	W =  -167.364 deg,	P =     0.000 deg,	R =   160.069 deg
};
P[589]{
   GP1:
	UF : 7, UT : 3,	CONFIG : 'F U T, 0, 0, 0',
	X =   227.898  mm,	Y =   288.444  mm,	Z =     0.000  mm,
	W =  -167.364 deg,	P =     0.000 deg,	R =   156.720 deg
};
P[590]{
   GP1:
	UF : 7, UT : 3,	CONFIG : 'F U T, 0, 0, 0',
	X =   244.343  mm,	Y =   274.653  mm,	Z =     0.000  mm,
	W =  -167.364 deg,	P =     0.000 deg,	R =   153.437 deg
};
P[591]{
   GP1:
	UF : 7, UT : 3,	CONFIG : 'F U T, 0, 0, 0',
	X =   259.557  mm,	Y =   260.313  mm,	Z =     0.000  mm,
	W =  -167.364 deg,	P =     0.000 deg,	R =   150.058 deg
};
P[592]{
   GP1:
	UF : 7, UT : 3,	CONFIG : 'F U T, 0, 0, 0',
	X =   274.330  mm,	Y =   244.717  mm,	Z =     0.000  mm,
	W =  -167.364 deg,	P =     0.000 deg,	R =   146.765 deg
};
P[593]{
   GP1:
	UF : 7, UT : 3,	CONFIG : 'F U T, 0, 0, 0',
	X =   288.138  mm,	Y =   228.286  mm,	Z =     0.000  mm,
	W =  -167.364 deg,	P =     0.000 deg,	R =   143.500 deg
};
P[594]{
   GP1:
	UF : 7, UT : 3,	CONFIG : 'F U T, 0, 0, 0',
	X =   300.682  mm,	Y =   211.488  mm,	Z =     0.000  mm,
	W =  -167.364 deg,	P =     0.000 deg,	R =   140.109 deg
};
P[595]{
   GP1:
	UF : 7, UT : 3,	CONFIG : 'F U T, 0, 0, 0',
	X =   312.553  mm,	Y =   193.530  mm,	Z =     0.000  mm,
	W =  -167.364 deg,	P =     0.000 deg,	R =   136.840 deg
};
P[596]{
   GP1:
	UF : 7, UT : 3,	CONFIG : 'F U T, 0, 0, 0',
	X =   324.894  mm,	Y =   172.024  mm,	Z =     0.000  mm,
	W =  -167.364 deg,	P =     0.000 deg,	R =   133.574 deg
};
P[597]{
   GP1:
	UF : 7, UT : 3,	CONFIG : 'F U T, 0, 0, 0',
	X =   324.894  mm,	Y =   172.024  mm,	Z =     0.000  mm,
	W =  -167.364 deg,	P =     0.000 deg,	R =   133.574 deg
};
P[598]{
   GP1:
	UF : 7, UT : 3,	CONFIG : 'F U T, 0, 0, 0',
	X =   324.894  mm,	Y =   172.024  mm,	Z =     0.000  mm,
	W =  -167.364 deg,	P =     0.000 deg,	R =   133.574 deg
};
P[599]{
   GP1:
	UF : 7, UT : 3,	CONFIG : 'F U T, 0, 0, 0',
	X =   324.894  mm,	Y =   172.024  mm,	Z =     0.000  mm,
	W =  -167.364 deg,	P =     0.000 deg,	R =   133.574 deg
};
P[600]{
   GP1:
	UF : 7, UT : 3,	CONFIG : 'F U T, 0, 0, 0',
	X =   337.049  mm,	Y =   146.732  mm,	Z =     0.000  mm,
	W =  -167.364 deg,	P =     0.000 deg,	R =   128.925 deg
};
P[601]{
   GP1:
	UF : 7, UT : 3,	CONFIG : 'F U T, 0, 0, 0',
	X =   337.049  mm,	Y =   146.732  mm,	Z =     0.000  mm,
	W =  -167.364 deg,	P =     0.000 deg,	R =   128.925 deg
};
P[602]{
   GP1:
	UF : 7, UT : 3,	CONFIG : 'F U T, 0, 0, 0',
	X =   337.049  mm,	Y =   146.732  mm,	Z =     0.000  mm,
	W =  -167.364 deg,	P =     0.000 deg,	R =   128.925 deg
};
P[603]{
   GP1:
	UF : 7, UT : 3,	CONFIG : 'F U T, 0, 0, 0',
	X =   337.049  mm,	Y =   146.732  mm,	Z =     0.000  mm,
	W =  -167.364 deg,	P =     0.000 deg,	R =   128.925 deg
};
P[604]{
   GP1:
	UF : 7, UT : 3,	CONFIG : 'F U T, 0, 0, 0',
	X =   344.666  mm,	Y =   127.847  mm,	Z =     0.000  mm,
	W =  -167.364 deg,	P =     0.000 deg,	R =   125.426 deg
};
P[605]{
   GP1:
	UF : 7, UT : 3,	CONFIG : 'F U T, 0, 0, 0',
	X =   351.381  mm,	Y =   108.000  mm,	Z =     0.000  mm,
	W =  -167.364 deg,	P =     0.000 deg,	R =   122.111 deg
};
P[606]{
   GP1:
	UF : 7, UT : 3,	CONFIG : 'F U T, 0, 0, 0',
	X =   357.037  mm,	Y =    87.546  mm,	Z =     0.000  mm,
	W =  -167.364 deg,	P =     0.000 deg,	R =   118.781 deg
};
P[607]{
   GP1:
	UF : 7, UT : 3,	CONFIG : 'F U T, 0, 0, 0',
	X =   361.521  mm,	Y =    66.649  mm,	Z =     0.000  mm,
	W =  -167.364 deg,	P =     0.000 deg,	R =   115.527 deg
};
P[608]{
   GP1:
	UF : 7, UT : 3,	CONFIG : 'F U T, 0, 0, 0',
	X =   364.734  mm,	Y =    45.876  mm,	Z =     0.000  mm,
	W =  -167.364 deg,	P =     0.000 deg,	R =   112.211 deg
};
P[609]{
   GP1:
	UF : 7, UT : 3,	CONFIG : 'F U T, 0, 0, 0',
	X =   366.785  mm,	Y =    24.736  mm,	Z =     0.000  mm,
	W =  -167.364 deg,	P =     0.000 deg,	R =   108.928 deg
};
P[610]{
   GP1:
	UF : 7, UT : 3,	CONFIG : 'F U T, 0, 0, 0',
	X =   367.626  mm,	Y =     0.000  mm,	Z =     0.000  mm,
	W =  -167.364 deg,	P =    -0.001 deg,	R =   105.687 deg
};
P[611]{
   GP1:
	UF : 7, UT : 3,	CONFIG : 'F U T, 0, 0, 0',
	X =   367.626  mm,	Y =     0.000  mm,	Z =     0.000  mm,
	W =  -167.364 deg,	P =    -0.001 deg,	R =   105.687 deg
};
P[612]{
   GP1:
	UF : 7, UT : 3,	CONFIG : 'F U T, 0, 0, 0',
	X =   367.626  mm,	Y =     0.000  mm,	Z =     0.000  mm,
	W =  -167.364 deg,	P =    -0.001 deg,	R =   105.687 deg
};
P[613]{
   GP1:
	UF : 7, UT : 3,	CONFIG : 'F U T, 0, 0, 0',
	X =   367.626  mm,	Y =     0.000  mm,	Z =     0.000  mm,
	W =  -167.364 deg,	P =    -0.001 deg,	R =   105.687 deg
};
P[614]{
   GP1:
	UF : 7, UT : 3,	CONFIG : 'F U T, 0, 0, 0',
	X =   364.492  mm,	Y =     0.000  mm,	Z =     0.000  mm,
	W =  -167.364 deg,	P =    -0.001 deg,	R =   105.687 deg
};
P[615]{
   GP1:
	UF : 7, UT : 3,	CONFIG : 'F U T, 0, 0, 0',
	X =   364.492  mm,	Y =     0.000  mm,	Z =     0.000  mm,
	W =  -167.364 deg,	P =    -0.001 deg,	R =   105.687 deg
};
P[616]{
   GP1:
	UF : 7, UT : 3,	CONFIG : 'F U T, 0, 0, 0',
	X =   364.492  mm,	Y =     0.000  mm,	Z =     0.000  mm,
	W =  -167.364 deg,	P =    -0.001 deg,	R =   105.687 deg
};
P[617]{
   GP1:
	UF : 7, UT : 3,	CONFIG : 'F U T, 0, 0, 0',
	X =   364.492  mm,	Y =     0.000  mm,	Z =     0.000  mm,
	W =  -167.364 deg,	P =    -0.001 deg,	R =   105.687 deg
};
P[618]{
   GP1:
	UF : 7, UT : 3,	CONFIG : 'F U T, 0, 0, 0',
	X =   363.409  mm,	Y =    27.784  mm,	Z =     0.000  mm,
	W =  -167.364 deg,	P =     0.000 deg,	R =   109.464 deg
};
P[619]{
   GP1:
	UF : 7, UT : 3,	CONFIG : 'F U T, 0, 0, 0',
	X =   360.720  mm,	Y =    52.147  mm,	Z =     0.000  mm,
	W =  -167.364 deg,	P =     0.000 deg,	R =   113.255 deg
};
P[620]{
   GP1:
	UF : 7, UT : 3,	CONFIG : 'F U T, 0, 0, 0',
	X =   356.378  mm,	Y =    76.373  mm,	Z =     0.000  mm,
	W =  -167.364 deg,	P =     0.000 deg,	R =   117.079 deg
};
P[621]{
   GP1:
	UF : 7, UT : 3,	CONFIG : 'F U T, 0, 0, 0',
	X =   350.467  mm,	Y =   100.057  mm,	Z =     0.000  mm,
	W =  -167.364 deg,	P =     0.000 deg,	R =   120.908 deg
};
P[622]{
   GP1:
	UF : 7, UT : 3,	CONFIG : 'F U T, 0, 0, 0',
	X =   343.019  mm,	Y =   123.198  mm,	Z =     0.000  mm,
	W =  -167.364 deg,	P =     0.000 deg,	R =   124.786 deg
};
P[623]{
   GP1:
	UF : 7, UT : 3,	CONFIG : 'F U T, 0, 0, 0',
	X =   334.719  mm,	Y =   144.230  mm,	Z =     0.000  mm,
	W =  -167.363 deg,	P =     0.000 deg,	R =   129.012 deg
};
P[624]{
   GP1:
	UF : 7, UT : 3,	CONFIG : 'F U T, 0, 0, 0',
	X =   334.719  mm,	Y =   144.230  mm,	Z =     0.000  mm,
	W =  -167.363 deg,	P =     0.000 deg,	R =   129.012 deg
};
P[625]{
   GP1:
	UF : 7, UT : 3,	CONFIG : 'F U T, 0, 0, 0',
	X =   334.719  mm,	Y =   144.230  mm,	Z =     0.000  mm,
	W =  -167.363 deg,	P =     0.000 deg,	R =   129.012 deg
};
P[626]{
   GP1:
	UF : 7, UT : 3,	CONFIG : 'F U T, 0, 0, 0',
	X =   334.719  mm,	Y =   144.230  mm,	Z =     0.000  mm,
	W =  -167.363 deg,	P =     0.000 deg,	R =   129.012 deg
};
P[627]{
   GP1:
	UF : 7, UT : 3,	CONFIG : 'F U T, 0, 0, 0',
	X =   321.465  mm,	Y =   171.771  mm,	Z =     0.000  mm,
	W =  -167.364 deg,	P =     0.000 deg,	R =   133.569 deg
};
P[628]{
   GP1:
	UF : 7, UT : 3,	CONFIG : 'F U T, 0, 0, 0',
	X =   321.465  mm,	Y =   171.771  mm,	Z =     0.000  mm,
	W =  -167.364 deg,	P =     0.000 deg,	R =   133.569 deg
};
P[629]{
   GP1:
	UF : 7, UT : 3,	CONFIG : 'F U T, 0, 0, 0',
	X =   321.465  mm,	Y =   171.771  mm,	Z =     0.000  mm,
	W =  -167.364 deg,	P =     0.000 deg,	R =   133.569 deg
};
P[630]{
   GP1:
	UF : 7, UT : 3,	CONFIG : 'F U T, 0, 0, 0',
	X =   321.465  mm,	Y =   171.771  mm,	Z =     0.000  mm,
	W =  -167.364 deg,	P =     0.000 deg,	R =   133.569 deg
};
P[631]{
   GP1:
	UF : 7, UT : 3,	CONFIG : 'F U T, 0, 0, 0',
	X =   308.090  mm,	Y =   194.731  mm,	Z =     0.000  mm,
	W =  -167.364 deg,	P =     0.000 deg,	R =   137.369 deg
};
P[632]{
   GP1:
	UF : 7, UT : 3,	CONFIG : 'F U T, 0, 0, 0',
	X =   294.440  mm,	Y =   214.811  mm,	Z =     0.000  mm,
	W =  -167.364 deg,	P =     0.000 deg,	R =   141.169 deg
};
P[633]{
   GP1:
	UF : 7, UT : 3,	CONFIG : 'F U T, 0, 0, 0',
	X =   279.300  mm,	Y =   234.157  mm,	Z =     0.000  mm,
	W =  -167.364 deg,	P =     0.000 deg,	R =   144.932 deg
};
P[634]{
   GP1:
	UF : 7, UT : 3,	CONFIG : 'F U T, 0, 0, 0',
	X =   263.275  mm,	Y =   252.044  mm,	Z =     0.000  mm,
	W =  -167.364 deg,	P =     0.000 deg,	R =   148.783 deg
};
P[635]{
   GP1:
	UF : 7, UT : 3,	CONFIG : 'F U T, 0, 0, 0',
	X =   246.100  mm,	Y =   268.837  mm,	Z =     0.000  mm,
	W =  -167.364 deg,	P =     0.000 deg,	R =   152.622 deg
};
P[636]{
   GP1:
	UF : 7, UT : 3,	CONFIG : 'F U T, 0, 0, 0',
	X =   227.367  mm,	Y =   284.855  mm,	Z =     0.000  mm,
	W =  -167.364 deg,	P =     0.000 deg,	R =   156.387 deg
};
P[637]{
   GP1:
	UF : 7, UT : 3,	CONFIG : 'F U T, 0, 0, 0',
	X =   208.034  mm,	Y =   299.269  mm,	Z =     0.000  mm,
	W =  -167.364 deg,	P =     0.000 deg,	R =   160.228 deg
};
P[638]{
   GP1:
	UF : 7, UT : 3,	CONFIG : 'F U T, 0, 0, 0',
	X =   187.768  mm,	Y =   312.382  mm,	Z =     0.000  mm,
	W =  -167.364 deg,	P =     0.000 deg,	R =   164.041 deg
};
P[639]{
   GP1:
	UF : 7, UT : 3,	CONFIG : 'F U T, 0, 0, 0',
	X =   166.350  mm,	Y =   324.294  mm,	Z =     0.000  mm,
	W =  -167.364 deg,	P =     0.000 deg,	R =   167.801 deg
};
P[640]{
   GP1:
	UF : 7, UT : 3,	CONFIG : 'F U T, 0, 0, 0',
	X =   144.440  mm,	Y =   334.629  mm,	Z =     0.000  mm,
	W =  -167.364 deg,	P =     0.000 deg,	R =   171.634 deg
};
P[641]{
   GP1:
	UF : 7, UT : 3,	CONFIG : 'F U T, 0, 0, 0',
	X =   122.176  mm,	Y =   343.383  mm,	Z =     0.000  mm,
	W =  -167.364 deg,	P =     0.000 deg,	R =   175.499 deg
};
P[642]{
   GP1:
	UF : 7, UT : 3,	CONFIG : 'F U T, 0, 0, 0',
	X =    95.933  mm,	Y =   351.637  mm,	Z =     0.000  mm,
	W =  -167.363 deg,	P =     0.000 deg,	R =   179.207 deg
};
P[643]{
   GP1:
	UF : 7, UT : 3,	CONFIG : 'F U T, 0, 0, 0',
	X =    95.933  mm,	Y =   351.637  mm,	Z =     0.000  mm,
	W =  -167.363 deg,	P =     0.000 deg,	R =   179.207 deg
};
P[644]{
   GP1:
	UF : 7, UT : 3,	CONFIG : 'F U T, 0, 0, 0',
	X =    95.933  mm,	Y =   351.637  mm,	Z =     0.000  mm,
	W =  -167.363 deg,	P =     0.000 deg,	R =   179.207 deg
};
P[645]{
   GP1:
	UF : 7, UT : 3,	CONFIG : 'F U T, 0, 0, 0',
	X =    95.933  mm,	Y =   351.637  mm,	Z =     0.000  mm,
	W =  -167.363 deg,	P =     0.000 deg,	R =   179.207 deg
};
P[646]{
   GP1:
	UF : 7, UT : 3,	CONFIG : 'F U T, 0, 0, 0',
	X =    66.134  mm,	Y =   358.425  mm,	Z =     0.000  mm,
	W =  -167.363 deg,	P =     0.000 deg,	R =  -175.664 deg
};
P[647]{
   GP1:
	UF : 7, UT : 3,	CONFIG : 'F U T, 0, 0, 0',
	X =    66.134  mm,	Y =   358.425  mm,	Z =     0.000  mm,
	W =  -167.363 deg,	P =     0.000 deg,	R =  -175.664 deg
};
P[648]{
   GP1:
	UF : 7, UT : 3,	CONFIG : 'F U T, 0, 0, 0',
	X =    66.134  mm,	Y =   358.425  mm,	Z =     0.000  mm,
	W =  -167.363 deg,	P =     0.000 deg,	R =  -175.664 deg
};
P[649]{
   GP1:
	UF : 7, UT : 3,	CONFIG : 'F U T, 0, 0, 0',
	X =    66.134  mm,	Y =   358.425  mm,	Z =     0.000  mm,
	W =  -167.363 deg,	P =     0.000 deg,	R =  -175.664 deg
};
P[650]{
   GP1:
	UF : 7, UT : 3,	CONFIG : 'F U T, 0, 0, 0',
	X =    44.878  mm,	Y =   361.697  mm,	Z =     0.000  mm,
	W =  -167.363 deg,	P =     0.000 deg,	R =  -171.981 deg
};
P[651]{
   GP1:
	UF : 7, UT : 3,	CONFIG : 'F U T, 0, 0, 0',
	X =    22.763  mm,	Y =   363.765  mm,	Z =     0.000  mm,
	W =  -167.363 deg,	P =     0.000 deg,	R =  -168.457 deg
};
P[652]{
   GP1:
	UF : 7, UT : 3,	CONFIG : 'F U T, 0, 0, 0',
	X =     0.089  mm,	Y =   364.491  mm,	Z =     0.000  mm,
